KUKA KRL program: EPS_2_26115_ST7256_A_20260223020028.src

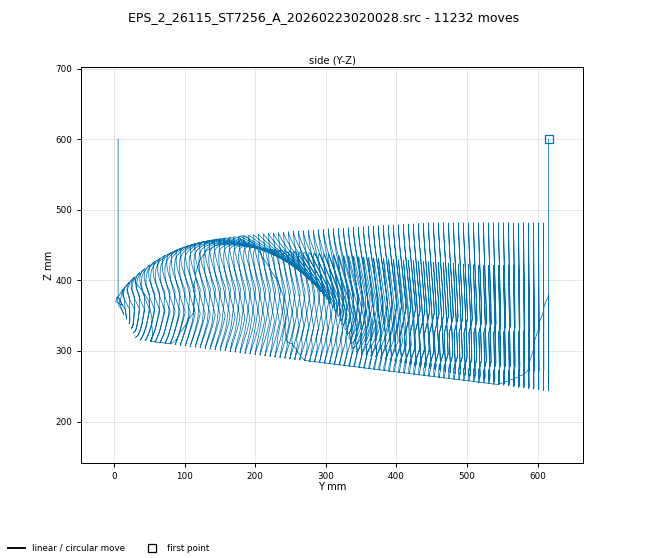
[picture p0: tool path of EPS_2_26115_ST7256_A_20260223020028.src, 11232 of 11234 moves have a stored position in this frame; points joined in program order, loops and branches not executed]
&ACCESS RVP
&REL 4
&COMMENT QRS 19112012
&PARAM EDITMASK = *
DEF PART()
EXT BAS (BAS_COMMAND :IN,REAL :IN )
INT I
BAS (#INITMOV,0 )

;KUKA QRS Post kuka4.cps  Date:22-06-2017 !

File_ID=3070

QRS_PRE_INIT()

;Init var - Until changes are made in qrs_pre_init
Outlet_Square_prg=0
Inlet_1_Square_prg=0
Inlet_2_Square_prg=0
Inlet_3_Square_prg=0
Inlet_4_Square_prg=0
Inlet_5_Square_prg=0

Outlet_1={X 0.000, Y 450.000, Z 332.000, B 0.000, E1 0.000 }
Inlet_1={X 0.000, Y 518.350, Z 272.000, B 0.000, E1 86.000 }
Outlet_1_type=299
Inlet_1_type=299
;QRS#1=Sidecore dimensions
;QRS#2=300-12" PVC SDR 35 Cut Back
;QRS#3=300-12" PVC SDR 35
;QRS#4=
;QRS#5=
;QRS#6=
;QRS#7=
;QRS#8=
;QRS#9=16M PSX
;QRS#10=16M PSX
;QRS#11=
;QRS#12=
;QRS#13=
;QRS#14=
;QRS#15=
;QRS#16=1220x127x762 2,5'
;QRS#17=EPS Height
;QRS#18=481,5
;QRS#19=*
;QRS#20= UPDATED VERSION 22-06-2017
;QRS#21=*
Outlet_Square=0150
Inlet_1_Square=0150
Inlet_2_Square=0
Inlet_3_Square=0
Inlet_4_Square=0
Inlet_5_Square=0
Mill_Square=1
Outlet_Square_Prg=216
Inlet_1_Square_prg=206

QRS_INIT()

$ADVANCE=5

; T1
PTP {E1 173.488,E2 173.488}
PTP {X 0,Y 615.495,A -85,B 0,C 180,E1 173.488,E2 173.488,E3 0,E4 0,E5 0,E6 0}
QRS_SPEED_INIT()
LIN {X 0,Y 615.495,Z 600,A -85,B 0,C 180,E1 173.488,E2 173.488,E3 0,E4 0,E5 0,E6 0} C_VEL
LIN {X 0,Y 615.495,Z 393.639,A -85,B 0,C 180,E1 173.488,E2 173.488} C_VEL
LIN {X 0,Y 615.495,Z 381.654,A -85,B 0,C 180,E1 173.488,E2 173.488} C_VEL
LIN {X 0,Y 615.494,Z 380.114,A -85,B 0,C 180,E1 173.42,E2 173.42} C_VEL
LIN {X 0,Y 615.498,Z 369.133,A -85,B 0,C 180,E1 172.289,E2 172.289} C_VEL
LIN {X 0,Y 615.497,Z 357.594,A -85,B 0,C 180,E1 171.298,E2 171.298} C_VEL
LIN {X 0,Y 615.497,Z 344.878,A -85,B 0,C 180,E1 170.387,E2 170.387} C_VEL
LIN {X 0,Y 615.489,Z 332.281,A -85,B 0,C 180,E1 169.639,E2 169.639} C_VEL
LIN {X 0,Y 615.455,Z 318.443,A -85,B 0,C 180,E1 168.968,E2 168.968} C_VEL
LIN {X 0,Y 615.481,Z 304.474,A -85,B 0,C 180,E1 168.431,E2 168.431} C_VEL
LIN {X 0,Y 615.493,Z 290.197,A -85,B 0,C 180,E1 168.014,E2 168.014} C_VEL
LIN {X 0,Y 615.498,Z 276.029,A -85,B 0,C 180,E1 167.721,E2 167.721} C_VEL
LIN {X 0,Y 615.488,Z 268.934,A -85,B 0,C 180,E1 167.616,E2 167.616} C_VEL
LIN {X 0,Y 615.468,Z 266.187,A -85,B 0,C 180,E1 165.45,E2 165.45} C_VEL
LIN {X 0,Y 615.461,Z 263.623,A -85,B 0,C 180,E1 163.412,E2 163.412} C_VEL
LIN {X 0,Y 615.456,Z 261.066,A -85,B 0,C 180,E1 161.353,E2 161.353} C_VEL
LIN {X 0,Y 615.452,Z 258.516,A -85,B 0,C 180,E1 159.268,E2 159.268} C_VEL
LIN {X 0,Y 615.452,Z 255.973,A -85,B 0,C 180,E1 157.154,E2 157.154} C_VEL
LIN {X 0,Y 615.492,Z 252.76,A -85,B 0,C 180,E1 154.431,E2 154.431} C_VEL
LIN {X 0,Y 615.451,Z 249.501,A -85,B 0,C 180,E1 151.557,E2 151.557} C_VEL
LIN {X 0,Y 615.49,Z 246.653,A -85,B 0,C 180,E1 148.914,E2 148.914} C_VEL
LIN {X 0,Y 615.496,Z 243.464,A -85,B 0,C 180,E1 145.978,E2 145.978} C_VEL
LIN {X 0,Y 615.445,Z 243.325,A -85,B 0,C 180,E1 143.572,E2 143.572} C_VEL
LIN {X 0,Y 615.497,Z 243.315,A -85,B 0,C 180,E1 140.937,E2 140.937} C_VEL
LIN {X 0,Y 615.489,Z 243.322,A -85,B 0,C 180,E1 138.526,E2 138.526} C_VEL
LIN {X 0,Y 615.45,Z 243.325,A -85,B 0,C 180,E1 135.847,E2 135.847} C_VEL
LIN {X 0,Y 615.489,Z 243.315,A -85,B 0,C 180,E1 133.047,E2 133.047} C_VEL
LIN {X 0,Y 615.477,Z 243.327,A -85,B 0,C 180,E1 130.608,E2 130.608} C_VEL
LIN {X 0,Y 615.465,Z 243.325,A -85,B 0,C 180,E1 128.009,E2 128.009} C_VEL
LIN {X 0,Y 615.476,Z 243.319,A -85,B 0,C 180,E1 125.617,E2 125.617} C_VEL
LIN {X 0,Y 615.485,Z 243.325,A -85,B 0,C 180,E1 123.237,E2 123.237} C_VEL
LIN {X 0,Y 615.47,Z 243.32,A -85,B 0,C 180,E1 120.921,E2 120.921} C_VEL
LIN {X 0,Y 615.488,Z 243.325,A -85,B 0,C 180,E1 118.45,E2 118.45} C_VEL
LIN {X 0,Y 615.474,Z 243.325,A -85,B 0,C 180,E1 115.716,E2 115.716} C_VEL
LIN {X 0,Y 615.477,Z 243.321,A -85,B 0,C 180,E1 112.845,E2 112.845} C_VEL
LIN {X 0,Y 615.465,Z 243.324,A -85,B 0,C 180,E1 110.55,E2 110.55} C_VEL
LIN {X 0,Y 615.492,Z 243.325,A -85,B 0,C 180,E1 107.957,E2 107.957} C_VEL
LIN {X 0,Y 615.484,Z 243.32,A -85,B 0,C 180,E1 105.226,E2 105.226} C_VEL
LIN {X 0,Y 615.446,Z 243.325,A -85,B 0,C 180,E1 102.531,E2 102.531} C_VEL
LIN {X 0,Y 615.497,Z 243.316,A -85,B 0,C 180,E1 99.862,E2 99.862} C_VEL
LIN {X 0,Y 615.485,Z 243.328,A -85,B 0,C 180,E1 97.216,E2 97.216} C_VEL
LIN {X 0,Y 615.459,Z 243.325,A -85,B 0,C 180,E1 94.585,E2 94.585} C_VEL
LIN {X 0,Y 615.5,Z 243.313,A -85,B 0,C 180,E1 91.963,E2 91.963} C_VEL
LIN {X 0,Y 615.468,Z 243.325,A -85,B 0,C 180,E1 89.346,E2 89.346} C_VEL
LIN {X 0,Y 615.476,Z 243.326,A -85,B 0,C 180,E1 86.727,E2 86.727} C_VEL
LIN {X 0,Y 615.498,Z 243.314,A -85,B 0,C 180,E1 84.101,E2 84.101} C_VEL
LIN {X 0,Y 615.451,Z 243.325,A -85,B 0,C 180,E1 81.463,E2 81.463} C_VEL
LIN {X 0,Y 615.492,Z 243.322,A -85,B 0,C 180,E1 78.807,E2 78.807} C_VEL
LIN {X 0,Y 615.493,Z 243.322,A -85,B 0,C 180,E1 76.066,E2 76.066} C_VEL
LIN {X 0,Y 615.453,Z 243.324,A -85,B 0,C 180,E1 73.412,E2 73.412} C_VEL
LIN {X 0,Y 615.486,Z 243.316,A -85,B 0,C 180,E1 70.662,E2 70.662} C_VEL
LIN {X 0,Y 615.456,Z 243.325,A -85,B 0,C 180,E1 67.862,E2 67.862} C_VEL
LIN {X 0,Y 615.465,Z 243.322,A -85,B 0,C 180,E1 65.727,E2 65.727} C_VEL
LIN {X 0,Y 615.481,Z 243.324,A -85,B 0,C 180,E1 63.555,E2 63.555} C_VEL
LIN {X 0,Y 615.447,Z 243.325,A -85,B 0,C 180,E1 61.34,E2 61.34} C_VEL
LIN {X 0,Y 615.495,Z 243.319,A -85,B 0,C 180,E1 58.913,E2 58.913} C_VEL
LIN {X 0,Y 615.491,Z 243.318,A -85,B 0,C 180,E1 56.466,E2 56.466} C_VEL
LIN {X 0,Y 615.453,Z 243.325,A -85,B 0,C 180,E1 53.572,E2 53.572} C_VEL
LIN {X 0,Y 615.496,Z 243.314,A -85,B 0,C 180,E1 50.937,E2 50.937} C_VEL
LIN {X 0,Y 615.495,Z 243.326,A -85,B 0,C 180,E1 48.526,E2 48.526} C_VEL
LIN {X 0,Y 615.46,Z 243.325,A -85,B 0,C 180,E1 45.847,E2 45.847} C_VEL
LIN {X 0,Y 615.489,Z 243.316,A -85,B 0,C 180,E1 43.047,E2 43.047} C_VEL
LIN {X 0,Y 615.467,Z 243.325,A -85,B 0,C 180,E1 40.608,E2 40.608} C_VEL
LIN {X 0,Y 615.479,Z 243.325,A -85,B 0,C 180,E1 38.01,E2 38.01} C_VEL
LIN {X 0,Y 615.47,Z 243.32,A -85,B 0,C 180,E1 35.617,E2 35.617} C_VEL
LIN {X 0,Y 615.482,Z 243.328,A -85,B 0,C 180,E1 33.237,E2 33.237} C_VEL
LIN {X 0,Y 615.476,Z 243.318,A -85,B 0,C 180,E1 30.921,E2 30.921} C_VEL
LIN {X 0,Y 615.474,Z 243.324,A -85,B 0,C 180,E1 28.447,E2 28.447} C_VEL
LIN {X 0,Y 615.498,Z 243.323,A -85,B 0,C 180,E1 25.57,E2 25.57} C_VEL
LIN {X 0,Y 615.485,Z 243.322,A -85,B 0,C 180,E1 22.845,E2 22.845} C_VEL
LIN {X 0,Y 615.448,Z 243.326,A -85,B 0,C 180,E1 20.546,E2 20.546} C_VEL
LIN {X 0,Y 615.493,Z 243.324,A -85,B 0,C 180,E1 17.957,E2 17.957} C_VEL
LIN {X 0,Y 615.489,Z 243.321,A -85,B 0,C 180,E1 15.226,E2 15.226} C_VEL
LIN {X 0,Y 615.45,Z 243.325,A -85,B 0,C 180,E1 12.531,E2 12.531} C_VEL
LIN {X 0,Y 615.496,Z 243.314,A -85,B 0,C 180,E1 9.862,E2 9.862} C_VEL
LIN {X 0,Y 615.476,Z 243.326,A -85,B 0,C 180,E1 7.216,E2 7.216} C_VEL
LIN {X 0,Y 615.471,Z 243.325,A -85,B 0,C 180,E1 4.585,E2 4.585} C_VEL
LIN {X 0,Y 615.5,Z 243.313,A -85,B 0,C 180,E1 1.963,E2 1.963} C_VEL
LIN {X 0,Y 615.456,Z 243.325,A -85,B 0,C 180,E1 -0.654,E2 -0.654} C_VEL
LIN {X 0,Y 615.488,Z 243.328,A -85,B 0,C 180,E1 -3.273,E2 -3.273} C_VEL
LIN {X 0,Y 615.499,Z 243.316,A -85,B 0,C 180,E1 -5.898,E2 -5.898} C_VEL
LIN {X 0,Y 615.446,Z 243.325,A -85,B 0,C 180,E1 -8.537,E2 -8.537} C_VEL
LIN {X 0,Y 615.484,Z 243.321,A -85,B 0,C 180,E1 -11.193,E2 -11.193} C_VEL
LIN {X 0,Y 615.498,Z 243.325,A -85,B 0,C 180,E1 -13.935,E2 -13.935} C_VEL
LIN {X 0,Y 615.466,Z 243.324,A -85,B 0,C 180,E1 -16.587,E2 -16.587} C_VEL
LIN {X 0,Y 615.482,Z 243.317,A -85,B 0,C 180,E1 -19.338,E2 -19.338} C_VEL
LIN {X 0,Y 615.448,Z 243.325,A -85,B 0,C 180,E1 -22.138,E2 -22.138} C_VEL
LIN {X 0,Y 615.477,Z 243.322,A -85,B 0,C 180,E1 -24.272,E2 -24.272} C_VEL
LIN {X 0,Y 615.468,Z 243.321,A -85,B 0,C 180,E1 -27.041,E2 -27.041} C_VEL
LIN {X 0,Y 615.464,Z 243.321,A -85,B 0,C 180,E1 -29.79,E2 -29.79} C_VEL
LIN {X 0,Y 615.481,Z 243.323,A -85,B 0,C 180,E1 -32.458,E2 -32.458} C_VEL
LIN {X 0,Y 615.459,Z 243.325,A -85,B 0,C 180,E1 -34.817,E2 -34.817} C_VEL
LIN {X 0,Y 615.492,Z 243.316,A -85,B 0,C 180,E1 -37.242,E2 -37.242} C_VEL
LIN {X 0,Y 615.474,Z 243.324,A -85,B 0,C 180,E1 -40.087,E2 -40.087} C_VEL
LIN {X 0,Y 615.451,Z 243.325,A -85,B 0,C 180,E1 -42.356,E2 -42.356} C_VEL
LIN {X 0,Y 615.491,Z 243.315,A -85,B 0,C 180,E1 -45.068,E2 -45.068} C_VEL
LIN {X 0,Y 615.454,Z 243.325,A -85,B 0,C 180,E1 -47.923,E2 -47.923} C_VEL
LIN {X 0,Y 615.474,Z 243.517,A -85,B 0,C 180,E1 -48.715,E2 -48.715} C_VEL
LIN {X 0,Y 615.44,Z 251.638,A -85,B 0,C 180,E1 -51.511,E2 -51.511} C_VEL
LIN {X 0,Y 615.45,Z 257.822,A -85,B 0,C 180,E1 -53.572,E2 -53.572} C_VEL
LIN {X 0,Y 615.483,Z 265.237,A -85,B 0,C 180,E1 -55.977,E2 -55.977} C_VEL
LIN {X 0,Y 615.485,Z 274.588,A -85,B 0,C 180,E1 -58.914,E2 -58.914} C_VEL
LIN {X 0,Y 615.486,Z 283.218,A -85,B 0,C 180,E1 -61.55,E2 -61.55} C_VEL
LIN {X 0,Y 615.472,Z 292.408,A -85,B 0,C 180,E1 -64.283,E2 -64.283} C_VEL
LIN {X 0,Y 615.455,Z 302.27,A -85,B 0,C 180,E1 -67.154,E2 -67.154} C_VEL
LIN {X 0,Y 615.425,Z 310.351,A -85,B 0,C 180,E1 -69.459,E2 -69.459} C_VEL
LIN {X 0,Y 615.486,Z 319.519,A -85,B 0,C 180,E1 -72.043,E2 -72.043} C_VEL
LIN {X 0,Y 615.465,Z 325.159,A -85,B 0,C 180,E1 -73.609,E2 -73.609} C_VEL
LIN {X 0,Y 615.49,Z 343.311,A -85,B 0,C 180,E1 -73.901,E2 -73.901} C_VEL
LIN {X 0,Y 615.497,Z 357.798,A -85,B 0,C 180,E1 -74.265,E2 -74.265} C_VEL
LIN {X 0,Y 615.463,Z 372.664,A -85,B 0,C 180,E1 -74.773,E2 -74.773} C_VEL
LIN {X 0,Y 615.468,Z 386.103,A -85,B 0,C 180,E1 -75.366,E2 -75.366} C_VEL
LIN {X 0,Y 615.498,Z 400.008,A -85,B 0,C 180,E1 -76.126,E2 -76.126} C_VEL
LIN {X 0,Y 615.496,Z 412.63,A -85,B 0,C 180,E1 -76.967,E2 -76.967} C_VEL
LIN {X 0,Y 615.496,Z 423.227,A -85,B 0,C 180,E1 -77.805,E2 -77.805} C_VEL
LIN {X 0,Y 615.496,Z 433.973,A -85,B 0,C 180,E1 -78.807,E2 -78.807} C_VEL
LIN {X 0,Y 615.496,Z 444.421,A -85,B 0,C 180,E1 -79.972,E2 -79.972} C_VEL
LIN {X 0,Y 615.496,Z 453.101,A -85,B 0,C 180,E1 -81.132,E2 -81.132} C_VEL
LIN {X 0,Y 615.494,Z 461.224,A -85,B 0,C 180,E1 -82.454,E2 -82.454} C_VEL
LIN {X 0,Y 615.496,Z 467.729,A -85,B 0,C 180,E1 -83.773,E2 -83.773} C_VEL
LIN {X 0,Y 615.496,Z 472.809,A -85,B 0,C 180,E1 -85.087,E2 -85.087} C_VEL
LIN {X 0,Y 615.495,Z 475.74,A -85,B 0,C 180,E1 -86.071,E2 -86.071} C_VEL
LIN {X 0,Y 615.494,Z 478.6,A -85,B 0,C 180,E1 -87.382,E2 -87.382} C_VEL
LIN {X 0,Y 615.492,Z 480.307,A -85,B 0,C 180,E1 -88.691,E2 -88.691} C_VEL
LIN {X 0,Y 615.491,Z 480.889,A -85,B 0,C 180,E1 -90,E2 -90} C_VEL
LIN {X 0,Y 615.492,Z 480.307,A -85,B 0,C 180,E1 -91.309,E2 -91.309} C_VEL
LIN {X 0,Y 615.494,Z 478.6,A -85,B 0,C 180,E1 -92.618,E2 -92.618} C_VEL
LIN {X 0,Y 615.495,Z 475.74,A -85,B 0,C 180,E1 -93.928,E2 -93.928} C_VEL
LIN {X 0,Y 615.491,Z 471.666,A -85,B 0,C 180,E1 -95.241,E2 -95.241} C_VEL
LIN {X 0,Y 615.49,Z 466.159,A -85,B 0,C 180,E1 -96.58,E2 -96.58} C_VEL
LIN {X 0,Y 615.493,Z 459.393,A -85,B 0,C 180,E1 -97.876,E2 -97.876} C_VEL
LIN {X 0,Y 615.495,Z 450.808,A -85,B 0,C 180,E1 -99.199,E2 -99.199} C_VEL
LIN {X 0,Y 615.494,Z 441.666,A -85,B 0,C 180,E1 -100.361,E2 -100.361} C_VEL
LIN {X 0,Y 615.497,Z 432.353,A -85,B 0,C 180,E1 -101.36,E2 -101.36} C_VEL
LIN {X 0,Y 615.496,Z 421.292,A -85,B 0,C 180,E1 -102.363,E2 -102.363} C_VEL
LIN {X 0,Y 615.498,Z 409.151,A -85,B 0,C 180,E1 -103.285,E2 -103.285} C_VEL
LIN {X 0,Y 615.498,Z 396.404,A -85,B 0,C 180,E1 -104.09,E2 -104.09} C_VEL
LIN {X 0,Y 615.46,Z 382.609,A -85,B 0,C 180,E1 -104.803,E2 -104.803} C_VEL
LIN {X 0,Y 615.474,Z 368.18,A -85,B 0,C 180,E1 -105.396,E2 -105.396} C_VEL
LIN {X 0,Y 615.496,Z 353.245,A -85,B 0,C 180,E1 -105.863,E2 -105.863} C_VEL
LIN {X 0,Y 615.483,Z 338.115,A -85,B 0,C 180,E1 -106.196,E2 -106.196} C_VEL
LIN {X 0,Y 615.465,Z 325.159,A -85,B 0,C 180,E1 -106.391,E2 -106.391} C_VEL
LIN {X 0,Y 615.433,Z 317.07,A -85,B 0,C 180,E1 -108.648,E2 -108.648} C_VEL
LIN {X 0,Y 615.498,Z 307.197,A -85,B 0,C 180,E1 -111.432,E2 -111.432} C_VEL
LIN {X 0,Y 615.446,Z 297.341,A -85,B 0,C 180,E1 -114.274,E2 -114.274} C_VEL
LIN {X 0,Y 615.491,Z 287.908,A -85,B 0,C 180,E1 -117.046,E2 -117.046} C_VEL
LIN {X 0,Y 615.477,Z 278.794,A -85,B 0,C 180,E1 -119.793,E2 -119.793} C_VEL
LIN {X 0,Y 615.476,Z 270.181,A -85,B 0,C 180,E1 -122.458,E2 -122.458} C_VEL
LIN {X 0,Y 615.493,Z 261.529,A -85,B 0,C 180,E1 -125.214,E2 -125.214} C_VEL
LIN {X 0,Y 615.446,Z 253.069,A -85,B 0,C 180,E1 -128.007,E2 -128.007} C_VEL
LIN {X 0,Y 615.427,Z 246.977,A -85,B 0,C 180,E1 -130.082,E2 -130.082} C_VEL
LIN {X 0,Y 615.46,Z 243.324,A -85,B 0,C 180,E1 -131.381,E2 -131.381} C_VEL
LIN {X 0,Y 615.44,Z 243.322,A -85,B 0,C 180,E1 -133.993,E2 -133.993} C_VEL
LIN {X 0,Y 615.456,Z 243.322,A -85,B 0,C 180,E1 -136.006,E2 -136.006} C_VEL
LIN {X 0,Y 615.467,Z 243.321,A -85,B 0,C 180,E1 -137.922,E2 -137.922} C_VEL
LIN {X 0,Y 615.493,Z 246.192,A -85,B 0,C 180,E1 -140.25,E2 -140.25} C_VEL
LIN {X 0,Y 615.487,Z 249.063,A -85,B 0,C 180,E1 -143.064,E2 -143.064} C_VEL
LIN {X 0,Y 615.458,Z 251.362,A -85,B 0,C 180,E1 -145.304,E2 -145.304} C_VEL
LIN {X 0,Y 615.461,Z 254.12,A -85,B 0,C 180,E1 -147.674,E2 -147.674} C_VEL
LIN {X 0,Y 615.489,Z 257.579,A -85,B 0,C 180,E1 -150.594,E2 -150.594} C_VEL
LIN {X 0,Y 615.465,Z 260.463,A -85,B 0,C 180,E1 -152.96,E2 -152.96} C_VEL
LIN {X 0,Y 615.481,Z 263.903,A -85,B 0,C 180,E1 -155.728,E2 -155.728} C_VEL
LIN {X 0,Y 615.49,Z 267.47,A -85,B 0,C 180,E1 -158.568,E2 -158.568} C_VEL
LIN {X 0,Y 615.483,Z 268.939,A -85,B 0,C 180,E1 -159.709,E2 -159.709} C_VEL
LIN {X 0,Y 615.491,Z 284.345,A -85,B 0,C 180,E1 -159.967,E2 -159.967} C_VEL
LIN {X 0,Y 615.489,Z 299.504,A -85,B 0,C 180,E1 -160.359,E2 -160.359} C_VEL
LIN {X 0,Y 615.464,Z 314.236,A -85,B 0,C 180,E1 -160.878,E2 -160.878} C_VEL
LIN {X 0,Y 615.481,Z 329.195,A -85,B 0,C 180,E1 -161.563,E2 -161.563} C_VEL
LIN {X 0,Y 615.498,Z 342.188,A -85,B 0,C 180,E1 -162.301,E2 -162.301} C_VEL
LIN {X 0,Y 615.496,Z 354.643,A -85,B 0,C 180,E1 -163.158,E2 -163.158} C_VEL
LIN {X 0,Y 615.496,Z 366.064,A -85,B 0,C 180,E1 -164.095,E2 -164.095} C_VEL
LIN {X 0,Y 615.494,Z 376.512,A -85,B 0,C 180,E1 -165.113,E2 -165.113} C_VEL
LIN {X 0,Y 615.493,Z 386.686,A -85,B 0,C 180,E1 -166.294,E2 -166.294} C_VEL
LIN {X 0,Y 615.493,Z 395.074,A -85,B 0,C 180,E1 -167.47,E2 -167.47} C_VEL
LIN {X 0,Y 615.495,Z 402.907,A -85,B 0,C 180,E1 -168.807,E2 -168.807} C_VEL
LIN {X 0,Y 615.498,Z 409.106,A -85,B 0,C 180,E1 -170.138,E2 -170.138} C_VEL
LIN {X 0,Y 615.491,Z 413.87,A -85,B 0,C 180,E1 -171.464,E2 -171.464} C_VEL
LIN {X 0,Y 615.493,Z 417.345,A -85,B 0,C 180,E1 -172.785,E2 -172.785} C_VEL
LIN {X 0,Y 615.499,Z 419.616,A -85,B 0,C 180,E1 -174.102,E2 -174.102} C_VEL
LIN {X 0,Y 615.497,Z 420.745,A -85,B 0,C 180,E1 -175.416,E2 -175.416} C_VEL
LIN {X 0,Y 615.491,Z 420.734,A -85,B 0,C 180,E1 -176.727,E2 -176.727} C_VEL
LIN {X 0,Y 615.5,Z 419.559,A -85,B 0,C 180,E1 -178.037,E2 -178.037} C_VEL
LIN {X 0,Y 615.491,Z 417.258,A -85,B 0,C 180,E1 -179.346,E2 -179.346} C_VEL
LIN {X 0,Y 615.49,Z 413.781,A -85,B 0,C 180,E1 -180.654,E2 -180.654} C_VEL
LIN {X 0,Y 615.5,Z 409.056,A -85,B 0,C 180,E1 -181.963,E2 -181.963} C_VEL
LIN {X 0,Y 615.492,Z 402.961,A -85,B 0,C 180,E1 -183.273,E2 -183.273} C_VEL
LIN {X 0,Y 615.494,Z 395.311,A -85,B 0,C 180,E1 -184.585,E2 -184.585} C_VEL
LIN {X 0,Y 615.495,Z 387.166,A -85,B 0,C 180,E1 -185.734,E2 -185.734} C_VEL
LIN {X 0,Y 615.494,Z 380.114,A -85,B 0,C 180,E1 -186.58,E2 -186.58} C_VEL
LIN {X 0,Y 614.823,Z 376.463,A -85,B 0,C 180,E1 -187.003,E2 -187.003} C_VEL
LIN {X 0,Y 611.954,Z 370.281,A -85,B 0,C 180,E1 -187.683,E2 -187.683} C_VEL
LIN {X 0,Y 609.129,Z 363.784,A -85,B 0,C 180,E1 -188.335,E2 -188.335} C_VEL
LIN {X 0,Y 608.527,Z 359.446,A -85,B 0,C 180,E1 -188.708,E2 -188.708} C_VEL
LIN {X 0,Y 608.536,Z 346.882,A -85,B 0,C 180,E1 -189.64,E2 -189.64} C_VEL
LIN {X 0,Y 608.57,Z 333.16,A -85,B 0,C 180,E1 -190.48,E2 -190.48} C_VEL
LIN {X 0,Y 608.559,Z 318.892,A -85,B 0,C 180,E1 -191.187,E2 -191.187} C_VEL
LIN {X 0,Y 608.62,Z 304.623,A -85,B 0,C 180,E1 -191.743,E2 -191.743} C_VEL
LIN {X 0,Y 608.667,Z 289.52,A -85,B 0,C 180,E1 -192.186,E2 -192.186} C_VEL
LIN {X 0,Y 608.694,Z 274.921,A -85,B 0,C 180,E1 -192.482,E2 -192.482} C_VEL
LIN {X 0,Y 608.431,Z 269.386,A -85,B 0,C 180,E1 -192.572,E2 -192.572} C_VEL
LIN {X 0,Y 608.399,Z 266.664,A -85,B 0,C 180,E1 -194.723,E2 -194.723} C_VEL
LIN {X 0,Y 608.399,Z 264.085,A -85,B 0,C 180,E1 -196.786,E2 -196.786} C_VEL
LIN {X 0,Y 608.409,Z 260.656,A -85,B 0,C 180,E1 -199.572,E2 -199.572} C_VEL
LIN {X 0,Y 608.398,Z 257.178,A -85,B 0,C 180,E1 -202.461,E2 -202.461} C_VEL
LIN {X 0,Y 608.404,Z 254.689,A -85,B 0,C 180,E1 -204.573,E2 -204.573} C_VEL
LIN {X 0,Y 608.416,Z 251.668,A -85,B 0,C 180,E1 -207.195,E2 -207.195} C_VEL
LIN {X 0,Y 608.422,Z 248.679,A -85,B 0,C 180,E1 -209.963,E2 -209.963} C_VEL
LIN {X 0,Y 608.436,Z 245.927,A -85,B 0,C 180,E1 -212.518,E2 -212.518} C_VEL
LIN {X 0,Y 608.452,Z 244.611,A -85,B 0,C 180,E1 -213.731,E2 -213.731} C_VEL
LIN {X 0,Y 608.44,Z 244.321,A -85,B 0,C 180,E1 -215.278,E2 -215.278} C_VEL
LIN {X 0,Y 608.449,Z 244.317,A -85,B 0,C 180,E1 -217.748,E2 -217.748} C_VEL
LIN {X 0,Y 608.453,Z 244.32,A -85,B 0,C 180,E1 -220.329,E2 -220.329} C_VEL
LIN {X 0,Y 608.477,Z 244.318,A -85,B 0,C 180,E1 -223.309,E2 -223.309} C_VEL
LIN {X 0,Y 608.464,Z 244.32,A -85,B 0,C 180,E1 -226.13,E2 -226.13} C_VEL
LIN {X 0,Y 608.454,Z 244.318,A -85,B 0,C 180,E1 -228.823,E2 -228.823} C_VEL
LIN {X 0,Y 608.449,Z 244.318,A -85,B 0,C 180,E1 -231.762,E2 -231.762} C_VEL
LIN {X 0,Y 608.447,Z 244.322,A -85,B 0,C 180,E1 -233.955,E2 -233.955} C_VEL
LIN {X 0,Y 608.446,Z 244.318,A -85,B 0,C 180,E1 -236.328,E2 -236.328} C_VEL
LIN {X 0,Y 608.448,Z 244.32,A -85,B 0,C 180,E1 -238.733,E2 -238.733} C_VEL
LIN {X 0,Y 608.473,Z 244.32,A -85,B 0,C 180,E1 -241.381,E2 -241.381} C_VEL
LIN {X 0,Y 608.425,Z 244.321,A -85,B 0,C 180,E1 -243.963,E2 -243.963} C_VEL
LIN {X 0,Y 608.449,Z 244.317,A -85,B 0,C 180,E1 -246.876,E2 -246.876} C_VEL
LIN {X 0,Y 608.454,Z 244.319,A -85,B 0,C 180,E1 -249.326,E2 -249.326} C_VEL
LIN {X 0,Y 608.439,Z 244.321,A -85,B 0,C 180,E1 -251.828,E2 -251.828} C_VEL
LIN {X 0,Y 608.47,Z 244.315,A -85,B 0,C 180,E1 -254.594,E2 -254.594} C_VEL
LIN {X 0,Y 608.422,Z 244.321,A -85,B 0,C 180,E1 -257.322,E2 -257.322} C_VEL
LIN {X 0,Y 608.462,Z 244.318,A -85,B 0,C 180,E1 -260.023,E2 -260.023} C_VEL
LIN {X 0,Y 608.465,Z 244.321,A -85,B 0,C 180,E1 -262.701,E2 -262.701} C_VEL
LIN {X 0,Y 608.426,Z 244.321,A -85,B 0,C 180,E1 -265.362,E2 -265.362} C_VEL
LIN {X 0,Y 608.47,Z 244.315,A -85,B 0,C 180,E1 -268.014,E2 -268.014} C_VEL
LIN {X 0,Y 608.465,Z 244.318,A -85,B 0,C 180,E1 -270.662,E2 -270.662} C_VEL
LIN {X 0,Y 608.471,Z 244.319,A -85,B 0,C 180,E1 -273.311,E2 -273.311} C_VEL
LIN {X 0,Y 608.471,Z 244.315,A -85,B 0,C 180,E1 -275.967,E2 -275.967} C_VEL
LIN {X 0,Y 608.427,Z 244.32,A -85,B 0,C 180,E1 -278.637,E2 -278.637} C_VEL
LIN {X 0,Y 608.482,Z 244.316,A -85,B 0,C 180,E1 -281.324,E2 -281.324} C_VEL
LIN {X 0,Y 608.473,Z 244.32,A -85,B 0,C 180,E1 -284.037,E2 -284.037} C_VEL
LIN {X 0,Y 608.432,Z 244.321,A -85,B 0,C 180,E1 -286.785,E2 -286.785} C_VEL
LIN {X 0,Y 608.454,Z 244.317,A -85,B 0,C 180,E1 -289.571,E2 -289.571} C_VEL
LIN {X 0,Y 608.433,Z 244.319,A -85,B 0,C 180,E1 -292.469,E2 -292.469} C_VEL
LIN {X 0,Y 608.453,Z 244.317,A -85,B 0,C 180,E1 -295.301,E2 -295.301} C_VEL
LIN {X 0,Y 608.446,Z 244.32,A -85,B 0,C 180,E1 -297.518,E2 -297.518} C_VEL
LIN {X 0,Y 608.441,Z 244.321,A -85,B 0,C 180,E1 -300.547,E2 -300.547} C_VEL
LIN {X 0,Y 608.463,Z 244.316,A -85,B 0,C 180,E1 -302.88,E2 -302.88} C_VEL
LIN {X 0,Y 608.43,Z 244.324,A -85,B 0,C 180,E1 -305.279,E2 -305.279} C_VEL
LIN {X 0,Y 608.459,Z 244.316,A -85,B 0,C 180,E1 -307.747,E2 -307.747} C_VEL
LIN {X 0,Y 608.446,Z 244.32,A -85,B 0,C 180,E1 -310.328,E2 -310.328} C_VEL
LIN {X 0,Y 608.445,Z 244.323,A -85,B 0,C 180,E1 -312.961,E2 -312.961} C_VEL
LIN {X 0,Y 608.454,Z 244.319,A -85,B 0,C 180,E1 -315.737,E2 -315.737} C_VEL
LIN {X 0,Y 608.453,Z 244.318,A -85,B 0,C 180,E1 -318.659,E2 -318.659} C_VEL
LIN {X 0,Y 608.46,Z 244.317,A -85,B 0,C 180,E1 -321.761,E2 -321.761} C_VEL
LIN {X 0,Y 608.446,Z 244.32,A -85,B 0,C 180,E1 -323.955,E2 -323.955} C_VEL
LIN {X 0,Y 608.448,Z 244.319,A -85,B 0,C 180,E1 -326.328,E2 -326.328} C_VEL
LIN {X 0,Y 608.451,Z 244.318,A -85,B 0,C 180,E1 -328.733,E2 -328.733} C_VEL
LIN {X 0,Y 608.47,Z 244.32,A -85,B 0,C 180,E1 -331.382,E2 -331.382} C_VEL
LIN {X 0,Y 608.432,Z 244.321,A -85,B 0,C 180,E1 -333.964,E2 -333.964} C_VEL
LIN {X 0,Y 608.473,Z 244.317,A -85,B 0,C 180,E1 -336.155,E2 -336.155} C_VEL
LIN {X 0,Y 608.447,Z 244.322,A -85,B 0,C 180,E1 -339.018,E2 -339.018} C_VEL
LIN {X 0,Y 608.442,Z 244.323,A -85,B 0,C 180,E1 -341.828,E2 -341.828} C_VEL
LIN {X 0,Y 608.473,Z 244.316,A -85,B 0,C 180,E1 -344.594,E2 -344.594} C_VEL
LIN {X 0,Y 608.421,Z 244.321,A -85,B 0,C 180,E1 -347.322,E2 -347.322} C_VEL
LIN {X 0,Y 608.465,Z 244.316,A -85,B 0,C 180,E1 -350.023,E2 -350.023} C_VEL
LIN {X 0,Y 608.444,Z 244.323,A -85,B 0,C 180,E1 -352.7,E2 -352.7} C_VEL
LIN {X 0,Y 608.437,Z 244.321,A -85,B 0,C 180,E1 -355.362,E2 -355.362} C_VEL
LIN {X 0,Y 608.469,Z 244.315,A -85,B 0,C 180,E1 -358.014,E2 -358.014} C_VEL
LIN {X 0,Y 608.454,Z 244.318,A -85,B 0,C 180,E1 -360.662,E2 -360.662} C_VEL
LIN {X 0,Y 608.482,Z 244.319,A -85,B 0,C 180,E1 -363.311,E2 -363.311} C_VEL
LIN {X 0,Y 608.469,Z 244.317,A -85,B 0,C 180,E1 -365.967,E2 -365.967} C_VEL
LIN {X 0,Y 608.426,Z 244.32,A -85,B 0,C 180,E1 -368.636,E2 -368.636} C_VEL
LIN {X 0,Y 608.462,Z 244.317,A -85,B 0,C 180,E1 -371.324,E2 -371.324} C_VEL
LIN {X 0,Y 608.475,Z 244.319,A -85,B 0,C 180,E1 -374.037,E2 -374.037} C_VEL
LIN {X 0,Y 608.438,Z 244.322,A -85,B 0,C 180,E1 -376.784,E2 -376.784} C_VEL
LIN {X 0,Y 608.451,Z 244.318,A -85,B 0,C 180,E1 -379.57,E2 -379.57} C_VEL
LIN {X 0,Y 608.433,Z 244.32,A -85,B 0,C 180,E1 -382.469,E2 -382.469} C_VEL
LIN {X 0,Y 608.449,Z 244.324,A -85,B 0,C 180,E1 -384.571,E2 -384.571} C_VEL
LIN {X 0,Y 608.471,Z 244.316,A -85,B 0,C 180,E1 -387.205,E2 -387.205} C_VEL
LIN {X 0,Y 608.43,Z 244.32,A -85,B 0,C 180,E1 -389.964,E2 -389.964} C_VEL
LIN {X 0,Y 608.458,Z 244.318,A -85,B 0,C 180,E1 -392.521,E2 -392.521} C_VEL
LIN {X 0,Y 608.424,Z 244.322,A -85,B 0,C 180,E1 -394.901,E2 -394.901} C_VEL
LIN {X 0,Y 608.467,Z 244.316,A -85,B 0,C 180,E1 -397.746,E2 -397.746} C_VEL
LIN {X 0,Y 608.435,Z 244.32,A -85,B 0,C 180,E1 -400.327,E2 -400.327} C_VEL
LIN {X 0,Y 608.467,Z 244.316,A -85,B 0,C 180,E1 -403.308,E2 -403.308} C_VEL
LIN {X 0,Y 608.473,Z 244.318,A -85,B 0,C 180,E1 -406.13,E2 -406.13} C_VEL
LIN {X 0,Y 608.44,Z 244.337,A -85,B 0,C 180,E1 -408.425,E2 -408.425} C_VEL
LIN {X 0,Y 608.541,Z 250.775,A -85,B 0,C 180,E1 -410.694,E2 -410.694} C_VEL
LIN {X 0,Y 608.507,Z 259.067,A -85,B 0,C 180,E1 -413.501,E2 -413.501} C_VEL
LIN {X 0,Y 608.519,Z 266.495,A -85,B 0,C 180,E1 -415.934,E2 -415.934} C_VEL
LIN {X 0,Y 608.491,Z 275.29,A -85,B 0,C 180,E1 -418.726,E2 -418.726} C_VEL
LIN {X 0,Y 608.499,Z 283.878,A -85,B 0,C 180,E1 -421.376,E2 -421.376} C_VEL
LIN {X 0,Y 608.447,Z 292.488,A -85,B 0,C 180,E1 -423.964,E2 -423.964} C_VEL
LIN {X 0,Y 608.472,Z 301.153,A -85,B 0,C 180,E1 -426.516,E2 -426.516} C_VEL
LIN {X 0,Y 608.42,Z 310.923,A -85,B 0,C 180,E1 -429.333,E2 -429.333} C_VEL
LIN {X 0,Y 608.45,Z 320.958,A -85,B 0,C 180,E1 -432.176,E2 -432.176} C_VEL
LIN {X 0,Y 608.426,Z 325.415,A -85,B 0,C 180,E1 -433.422,E2 -433.422} C_VEL
LIN {X 0,Y 608.682,Z 332.489,A -85,B 0,C 180,E1 -433.528,E2 -433.528} C_VEL
LIN {X 0,Y 608.675,Z 347.584,A -85,B 0,C 180,E1 -433.814,E2 -433.814} C_VEL
LIN {X 0,Y 608.623,Z 363.2,A -85,B 0,C 180,E1 -434.254,E2 -434.254} C_VEL
LIN {X 0,Y 608.573,Z 376.817,A -85,B 0,C 180,E1 -434.768,E2 -434.768} C_VEL
LIN {X 0,Y 608.565,Z 391.1,A -85,B 0,C 180,E1 -435.453,E2 -435.453} C_VEL
LIN {X 0,Y 608.558,Z 404.109,A -85,B 0,C 180,E1 -436.22,E2 -436.22} C_VEL
LIN {X 0,Y 608.518,Z 416.103,A -85,B 0,C 180,E1 -437.069,E2 -437.069} C_VEL
LIN {X 0,Y 608.509,Z 427.191,A -85,B 0,C 180,E1 -438.001,E2 -438.001} C_VEL
LIN {X 0,Y 608.477,Z 437.641,A -85,B 0,C 180,E1 -439.04,E2 -439.04} C_VEL
LIN {X 0,Y 608.471,Z 447.368,A -85,B 0,C 180,E1 -440.191,E2 -440.191} C_VEL
LIN {X 0,Y 608.467,Z 455.654,A -85,B 0,C 180,E1 -441.364,E2 -441.364} C_VEL
LIN {X 0,Y 608.456,Z 463.426,A -85,B 0,C 180,E1 -442.7,E2 -442.7} C_VEL
LIN {X 0,Y 608.437,Z 469.608,A -85,B 0,C 180,E1 -444.033,E2 -444.033} C_VEL
LIN {X 0,Y 608.427,Z 474.383,A -85,B 0,C 180,E1 -445.362,E2 -445.362} C_VEL
LIN {X 0,Y 608.421,Z 477.885,A -85,B 0,C 180,E1 -446.689,E2 -446.689} C_VEL
LIN {X 0,Y 608.444,Z 480.191,A -85,B 0,C 180,E1 -448.014,E2 -448.014} C_VEL
LIN {X 0,Y 608.434,Z 481.351,A -85,B 0,C 180,E1 -449.338,E2 -449.338} C_VEL
LIN {X 0,Y 608.434,Z 481.351,A -85,B 0,C 180,E1 -450.662,E2 -450.662} C_VEL
LIN {X 0,Y 608.444,Z 480.191,A -85,B 0,C 180,E1 -451.986,E2 -451.986} C_VEL
LIN {X 0,Y 608.421,Z 477.885,A -85,B 0,C 180,E1 -453.311,E2 -453.311} C_VEL
LIN {X 0,Y 608.427,Z 474.383,A -85,B 0,C 180,E1 -454.638,E2 -454.638} C_VEL
LIN {X 0,Y 608.437,Z 469.608,A -85,B 0,C 180,E1 -455.967,E2 -455.967} C_VEL
LIN {X 0,Y 608.456,Z 463.426,A -85,B 0,C 180,E1 -457.3,E2 -457.3} C_VEL
LIN {X 0,Y 608.467,Z 455.654,A -85,B 0,C 180,E1 -458.636,E2 -458.636} C_VEL
LIN {X 0,Y 608.471,Z 447.369,A -85,B 0,C 180,E1 -459.809,E2 -459.809} C_VEL
LIN {X 0,Y 608.492,Z 436.653,A -85,B 0,C 180,E1 -461.063,E2 -461.063} C_VEL
LIN {X 0,Y 608.522,Z 425.275,A -85,B 0,C 180,E1 -462.168,E2 -462.168} C_VEL
LIN {X 0,Y 608.547,Z 413.853,A -85,B 0,C 180,E1 -463.1,E2 -463.1} C_VEL
LIN {X 0,Y 608.563,Z 401.446,A -85,B 0,C 180,E1 -463.95,E2 -463.95} C_VEL
LIN {X 0,Y 608.576,Z 387.858,A -85,B 0,C 180,E1 -464.718,E2 -464.718} C_VEL
LIN {X 0,Y 608.593,Z 373.791,A -85,B 0,C 180,E1 -465.36,E2 -465.36} C_VEL
LIN {X 0,Y 608.643,Z 359.295,A -85,B 0,C 180,E1 -465.874,E2 -465.874} C_VEL
LIN {X 0,Y 608.675,Z 343.318,A -85,B 0,C 180,E1 -466.284,E2 -466.284} C_VEL
LIN {X 0,Y 608.671,Z 327.102,A -85,B 0,C 180,E1 -466.546,E2 -466.546} C_VEL
LIN {X 0,Y 608.433,Z 325.333,A -85,B 0,C 180,E1 -466.6,E2 -466.6} C_VEL
LIN {X 0,Y 608.435,Z 316.007,A -85,B 0,C 180,E1 -469.22,E2 -469.22} C_VEL
LIN {X 0,Y 608.445,Z 306.105,A -85,B 0,C 180,E1 -472.049,E2 -472.049} C_VEL
LIN {X 0,Y 608.439,Z 297.44,A -85,B 0,C 180,E1 -474.572,E2 -474.572} C_VEL
LIN {X 0,Y 608.484,Z 288.561,A -85,B 0,C 180,E1 -477.208,E2 -477.208} C_VEL
LIN {X 0,Y 608.484,Z 279.477,A -85,B 0,C 180,E1 -479.974,E2 -479.974} C_VEL
LIN {X 0,Y 608.516,Z 271.296,A -85,B 0,C 180,E1 -482.531,E2 -482.531} C_VEL
LIN {X 0,Y 608.553,Z 262.781,A -85,B 0,C 180,E1 -485.271,E2 -485.271} C_VEL
LIN {X 0,Y 608.532,Z 255.354,A -85,B 0,C 180,E1 -487.742,E2 -487.742} C_VEL
LIN {X 0,Y 608.517,Z 247.82,A -85,B 0,C 180,E1 -490.336,E2 -490.336} C_VEL
LIN {X 0,Y 608.426,Z 244.322,A -85,B 0,C 180,E1 -491.624,E2 -491.624} C_VEL
LIN {X 0,Y 608.425,Z 244.321,A -85,B 0,C 180,E1 -494.261,E2 -494.261} C_VEL
LIN {X 0,Y 608.45,Z 244.317,A -85,B 0,C 180,E1 -497.04,E2 -497.04} C_VEL
LIN {X 0,Y 608.448,Z 244.32,A -85,B 0,C 180,E1 -497.938,E2 -497.938} C_VEL
LIN {X 0,Y 608.45,Z 247.646,A -85,B 0,C 180,E1 -500.705,E2 -500.705} C_VEL
LIN {X 0,Y 608.447,Z 250.017,A -85,B 0,C 180,E1 -503.085,E2 -503.085} C_VEL
LIN {X 0,Y 608.396,Z 252.389,A -85,B 0,C 180,E1 -505.526,E2 -505.526} C_VEL
LIN {X 0,Y 608.404,Z 255.14,A -85,B 0,C 180,E1 -507.902,E2 -507.902} C_VEL
LIN {X 0,Y 608.444,Z 257.88,A -85,B 0,C 180,E1 -510.219,E2 -510.219} C_VEL
LIN {X 0,Y 608.418,Z 261.005,A -85,B 0,C 180,E1 -512.805,E2 -512.805} C_VEL
LIN {X 0,Y 608.412,Z 264.237,A -85,B 0,C 180,E1 -515.427,E2 -515.427} C_VEL
LIN {X 0,Y 608.416,Z 267.849,A -85,B 0,C 180,E1 -518.307,E2 -518.307} C_VEL
LIN {X 0,Y 608.409,Z 269.379,A -85,B 0,C 180,E1 -519.512,E2 -519.512} C_VEL
LIN {X 0,Y 608.671,Z 273.442,A -85,B 0,C 180,E1 -519.586,E2 -519.586} C_VEL
LIN {X 0,Y 608.655,Z 288.814,A -85,B 0,C 180,E1 -519.887,E2 -519.887} C_VEL
LIN {X 0,Y 608.656,Z 303.324,A -85,B 0,C 180,E1 -520.305,E2 -520.305} C_VEL
LIN {X 0,Y 608.585,Z 318.174,A -85,B 0,C 180,E1 -520.872,E2 -520.872} C_VEL
LIN {X 0,Y 608.581,Z 331.28,A -85,B 0,C 180,E1 -521.508,E2 -521.508} C_VEL
LIN {X 0,Y 608.542,Z 344.128,A -85,B 0,C 180,E1 -522.266,E2 -522.266} C_VEL
LIN {X 0,Y 608.532,Z 356.316,A -85,B 0,C 180,E1 -523.132,E2 -523.132} C_VEL
LIN {X 0,Y 608.503,Z 367.55,A -85,B 0,C 180,E1 -524.08,E2 -524.08} C_VEL
LIN {X 0,Y 608.486,Z 377.851,A -85,B 0,C 180,E1 -525.109,E2 -525.109} C_VEL
LIN {X 0,Y 608.473,Z 387.879,A -85,B 0,C 180,E1 -526.304,E2 -526.304} C_VEL
LIN {X 0,Y 608.464,Z 396.203,A -85,B 0,C 180,E1 -527.493,E2 -527.493} C_VEL
LIN {X 0,Y 608.458,Z 403.049,A -85,B 0,C 180,E1 -528.676,E2 -528.676} C_VEL
LIN {X 0,Y 608.437,Z 409.371,A -85,B 0,C 180,E1 -530.023,E2 -530.023} C_VEL
LIN {X 0,Y 608.423,Z 414.245,A -85,B 0,C 180,E1 -531.364,E2 -531.364} C_VEL
LIN {X 0,Y 608.423,Z 417.813,A -85,B 0,C 180,E1 -532.7,E2 -532.7} C_VEL
LIN {X 0,Y 608.435,Z 420.161,A -85,B 0,C 180,E1 -534.033,E2 -534.033} C_VEL
LIN {X 0,Y 608.43,Z 421.344,A -85,B 0,C 180,E1 -535.362,E2 -535.362} C_VEL
LIN {X 0,Y 608.416,Z 421.355,A -85,B 0,C 180,E1 -536.689,E2 -536.689} C_VEL
LIN {X 0,Y 608.445,Z 420.211,A -85,B 0,C 180,E1 -538.014,E2 -538.014} C_VEL
LIN {X 0,Y 608.435,Z 417.924,A -85,B 0,C 180,E1 -539.338,E2 -539.338} C_VEL
LIN {X 0,Y 608.434,Z 414.449,A -85,B 0,C 180,E1 -540.662,E2 -540.662} C_VEL
LIN {X 0,Y 608.445,Z 409.72,A -85,B 0,C 180,E1 -541.986,E2 -541.986} C_VEL
LIN {X 0,Y 608.433,Z 403.608,A -85,B 0,C 180,E1 -543.311,E2 -543.311} C_VEL
LIN {X 0,Y 608.462,Z 395.943,A -85,B 0,C 180,E1 -544.638,E2 -544.638} C_VEL
LIN {X 0,Y 608.477,Z 387.773,A -85,B 0,C 180,E1 -545.801,E2 -545.801} C_VEL
LIN {X 0,Y 608.49,Z 377.986,A -85,B 0,C 180,E1 -546.966,E2 -546.966} C_VEL
LIN {X 0,Y 608.491,Z 368.008,A -85,B 0,C 180,E1 -547.967,E2 -547.967} C_VEL
LIN {X 0,Y 608.527,Z 359.446,A -85,B 0,C 180,E1 -548.708,E2 -548.708} C_VEL
LIN {X 0,Y 607.933,Z 355.043,A -85,B 0,C 180,E1 -549.071,E2 -549.071} C_VEL
LIN {X 0,Y 605.145,Z 347.83,A -85,B 0,C 180,E1 -549.663,E2 -549.663} C_VEL
LIN {X 0,Y 602.323,Z 340.351,A -85,B 0,C 180,E1 -550.22,E2 -550.22} C_VEL
LIN {X 0,Y 601.669,Z 335.425,A -85,B 0,C 180,E1 -550.524,E2 -550.524} C_VEL
LIN {X 0,Y 601.69,Z 322.242,A -85,B 0,C 180,E1 -551.213,E2 -551.213} C_VEL
LIN {X 0,Y 601.763,Z 308.367,A -85,B 0,C 180,E1 -551.794,E2 -551.794} C_VEL
LIN {X 0,Y 601.849,Z 293.034,A -85,B 0,C 180,E1 -552.284,E2 -552.284} C_VEL
LIN {X 0,Y 601.871,Z 277.738,A -85,B 0,C 180,E1 -552.626,E2 -552.626} C_VEL
LIN {X 0,Y 601.644,Z 271.313,A -85,B 0,C 180,E1 -552.732,E2 -552.732} C_VEL
LIN {X 0,Y 601.324,Z 269.368,A -85,B 0,C 180,E1 -552.788,E2 -552.788} C_VEL
LIN {X 0,Y 601.297,Z 266.728,A -85,B 0,C 180,E1 -554.9,E2 -554.9} C_VEL
LIN {X 0,Y 601.323,Z 264.148,A -85,B 0,C 180,E1 -556.989,E2 -556.989} C_VEL
LIN {X 0,Y 601.311,Z 260.721,A -85,B 0,C 180,E1 -559.813,E2 -559.813} C_VEL
LIN {X 0,Y 601.317,Z 257.431,A -85,B 0,C 180,E1 -562.582,E2 -562.582} C_VEL
LIN {X 0,Y 601.333,Z 254.756,A -85,B 0,C 180,E1 -564.882,E2 -564.882} C_VEL
LIN {X 0,Y 601.337,Z 252.05,A -85,B 0,C 180,E1 -567.347,E2 -567.347} C_VEL
LIN {X 0,Y 601.343,Z 249.015,A -85,B 0,C 180,E1 -570.169,E2 -570.169} C_VEL
LIN {X 0,Y 601.363,Z 246.304,A -85,B 0,C 180,E1 -572.706,E2 -572.706} C_VEL
LIN {X 0,Y 601.372,Z 245.204,A -85,B 0,C 180,E1 -574.122,E2 -574.122} C_VEL
LIN {X 0,Y 601.397,Z 245.196,A -85,B 0,C 180,E1 -576.584,E2 -576.584} C_VEL
LIN {X 0,Y 601.418,Z 245.193,A -85,B 0,C 180,E1 -579.533,E2 -579.533} C_VEL
LIN {X 0,Y 601.417,Z 245.198,A -85,B 0,C 180,E1 -581.766,E2 -581.766} C_VEL
LIN {X 0,Y 601.402,Z 245.199,A -85,B 0,C 180,E1 -584.532,E2 -584.532} C_VEL
LIN {X 0,Y 601.418,Z 245.195,A -85,B 0,C 180,E1 -587.409,E2 -587.409} C_VEL
LIN {X 0,Y 601.382,Z 245.198,A -85,B 0,C 180,E1 -590.002,E2 -590.002} C_VEL
LIN {X 0,Y 601.439,Z 245.193,A -85,B 0,C 180,E1 -592.618,E2 -592.618} C_VEL
LIN {X 0,Y 601.417,Z 245.196,A -85,B 0,C 180,E1 -595.068,E2 -595.068} C_VEL
LIN {X 0,Y 601.401,Z 245.195,A -85,B 0,C 180,E1 -597.482,E2 -597.482} C_VEL
LIN {X 0,Y 601.433,Z 245.197,A -85,B 0,C 180,E1 -599.851,E2 -599.851} C_VEL
LIN {X 0,Y 601.421,Z 245.195,A -85,B 0,C 180,E1 -602.637,E2 -602.637} C_VEL
LIN {X 0,Y 601.39,Z 245.197,A -85,B 0,C 180,E1 -605.121,E2 -605.121} C_VEL
LIN {X 0,Y 601.42,Z 245.194,A -85,B 0,C 180,E1 -608.041,E2 -608.041} C_VEL
LIN {X 0,Y 601.41,Z 245.196,A -85,B 0,C 180,E1 -610.901,E2 -610.901} C_VEL
LIN {X 0,Y 601.443,Z 245.195,A -85,B 0,C 180,E1 -613.713,E2 -613.713} C_VEL
LIN {X 0,Y 601.414,Z 245.197,A -85,B 0,C 180,E1 -616.484,E2 -616.484} C_VEL
LIN {X 0,Y 601.388,Z 245.198,A -85,B 0,C 180,E1 -619.223,E2 -619.223} C_VEL
LIN {X 0,Y 601.443,Z 245.19,A -85,B 0,C 180,E1 -621.939,E2 -621.939} C_VEL
LIN {X 0,Y 601.407,Z 245.196,A -85,B 0,C 180,E1 -624.636,E2 -624.636} C_VEL
LIN {X 0,Y 601.445,Z 245.196,A -85,B 0,C 180,E1 -627.321,E2 -627.321} C_VEL
LIN {X 0,Y 601.449,Z 245.191,A -85,B 0,C 180,E1 -630,E2 -630} C_VEL
LIN {X 0,Y 601.415,Z 245.193,A -85,B 0,C 180,E1 -632.679,E2 -632.679} C_VEL
LIN {X 0,Y 601.428,Z 245.193,A -85,B 0,C 180,E1 -635.364,E2 -635.364} C_VEL
LIN {X 0,Y 601.437,Z 245.196,A -85,B 0,C 180,E1 -638.061,E2 -638.061} C_VEL
LIN {X 0,Y 601.421,Z 245.199,A -85,B 0,C 180,E1 -641.008,E2 -641.008} C_VEL
LIN {X 0,Y 601.414,Z 245.194,A -85,B 0,C 180,E1 -643.516,E2 -643.516} C_VEL
LIN {X 0,Y 601.406,Z 245.195,A -85,B 0,C 180,E1 -646.614,E2 -646.614} C_VEL
LIN {X 0,Y 601.422,Z 245.194,A -85,B 0,C 180,E1 -649.099,E2 -649.099} C_VEL
LIN {X 0,Y 601.396,Z 245.199,A -85,B 0,C 180,E1 -651.96,E2 -651.96} C_VEL
LIN {X 0,Y 601.4,Z 245.2,A -85,B 0,C 180,E1 -654.879,E2 -654.879} C_VEL
LIN {X 0,Y 601.413,Z 245.195,A -85,B 0,C 180,E1 -657.361,E2 -657.361} C_VEL
LIN {X 0,Y 601.402,Z 245.195,A -85,B 0,C 180,E1 -660.166,E2 -660.166} C_VEL
LIN {X 0,Y 601.428,Z 245.194,A -85,B 0,C 180,E1 -662.716,E2 -662.716} C_VEL
LIN {X 0,Y 601.383,Z 245.2,A -85,B 0,C 180,E1 -665.11,E2 -665.11} C_VEL
LIN {X 0,Y 601.437,Z 245.192,A -85,B 0,C 180,E1 -667.419,E2 -667.419} C_VEL
LIN {X 0,Y 601.407,Z 245.201,A -85,B 0,C 180,E1 -669.996,E2 -669.996} C_VEL
LIN {X 0,Y 601.379,Z 245.2,A -85,B 0,C 180,E1 -672.674,E2 -672.674} C_VEL
LIN {X 0,Y 601.431,Z 245.192,A -85,B 0,C 180,E1 -675.482,E2 -675.482} C_VEL
LIN {X 0,Y 601.418,Z 245.193,A -85,B 0,C 180,E1 -678.408,E2 -678.408} C_VEL
LIN {X 0,Y 601.413,Z 245.194,A -85,B 0,C 180,E1 -681.532,E2 -681.532} C_VEL
LIN {X 0,Y 601.4,Z 245.201,A -85,B 0,C 180,E1 -683.74,E2 -683.74} C_VEL
LIN {X 0,Y 601.406,Z 245.195,A -85,B 0,C 180,E1 -686.069,E2 -686.069} C_VEL
LIN {X 0,Y 601.417,Z 245.193,A -85,B 0,C 180,E1 -689.058,E2 -689.058} C_VEL
LIN {X 0,Y 601.43,Z 245.197,A -85,B 0,C 180,E1 -691.373,E2 -691.373} C_VEL
LIN {X 0,Y 601.41,Z 245.198,A -85,B 0,C 180,E1 -694.134,E2 -694.134} C_VEL
LIN {X 0,Y 601.403,Z 245.195,A -85,B 0,C 180,E1 -696.589,E2 -696.589} C_VEL
LIN {X 0,Y 601.405,Z 245.195,A -85,B 0,C 180,E1 -699.477,E2 -699.477} C_VEL
LIN {X 0,Y 601.393,Z 245.198,A -85,B 0,C 180,E1 -702.311,E2 -702.311} C_VEL
LIN {X 0,Y 601.417,Z 245.194,A -85,B 0,C 180,E1 -704.409,E2 -704.409} C_VEL
LIN {X 0,Y 601.375,Z 245.198,A -85,B 0,C 180,E1 -707.171,E2 -707.171} C_VEL
LIN {X 0,Y 601.44,Z 245.192,A -85,B 0,C 180,E1 -709.905,E2 -709.905} C_VEL
LIN {X 0,Y 601.411,Z 245.2,A -85,B 0,C 180,E1 -712.614,E2 -712.614} C_VEL
LIN {X 0,Y 601.406,Z 245.197,A -85,B 0,C 180,E1 -715.308,E2 -715.308} C_VEL
LIN {X 0,Y 601.438,Z 245.191,A -85,B 0,C 180,E1 -717.991,E2 -717.991} C_VEL
LIN {X 0,Y 601.428,Z 245.193,A -85,B 0,C 180,E1 -720.669,E2 -720.669} C_VEL
LIN {X 0,Y 601.433,Z 245.197,A -85,B 0,C 180,E1 -723.349,E2 -723.349} C_VEL
LIN {X 0,Y 601.418,Z 245.196,A -85,B 0,C 180,E1 -726.037,E2 -726.037} C_VEL
LIN {X 0,Y 601.393,Z 245.196,A -85,B 0,C 180,E1 -728.738,E2 -728.738} C_VEL
LIN {X 0,Y 601.428,Z 245.192,A -85,B 0,C 180,E1 -731.458,E2 -731.458} C_VEL
LIN {X 0,Y 601.417,Z 245.196,A -85,B 0,C 180,E1 -734.205,E2 -734.205} C_VEL
LIN {X 0,Y 601.414,Z 245.2,A -85,B 0,C 180,E1 -736.986,E2 -736.986} C_VEL
LIN {X 0,Y 601.402,Z 245.199,A -85,B 0,C 180,E1 -739.809,E2 -739.809} C_VEL
LIN {X 0,Y 601.405,Z 245.196,A -85,B 0,C 180,E1 -742.683,E2 -742.683} C_VEL
LIN {X 0,Y 601.402,Z 245.198,A -85,B 0,C 180,E1 -744.878,E2 -744.878} C_VEL
LIN {X 0,Y 601.408,Z 245.197,A -85,B 0,C 180,E1 -747.36,E2 -747.36} C_VEL
LIN {X 0,Y 601.403,Z 245.196,A -85,B 0,C 180,E1 -750.165,E2 -750.165} C_VEL
LIN {X 0,Y 601.421,Z 245.194,A -85,B 0,C 180,E1 -752.714,E2 -752.714} C_VEL
LIN {X 0,Y 601.375,Z 245.203,A -85,B 0,C 180,E1 -755.108,E2 -755.108} C_VEL
LIN {X 0,Y 601.438,Z 245.191,A -85,B 0,C 180,E1 -757.419,E2 -757.419} C_VEL
LIN {X 0,Y 601.415,Z 245.197,A -85,B 0,C 180,E1 -759.995,E2 -759.995} C_VEL
LIN {X 0,Y 601.384,Z 245.201,A -85,B 0,C 180,E1 -762.673,E2 -762.673} C_VEL
LIN {X 0,Y 601.429,Z 245.194,A -85,B 0,C 180,E1 -765.482,E2 -765.482} C_VEL
LIN {X 0,Y 601.434,Z 245.306,A -85,B 0,C 180,E1 -768.179,E2 -768.179} C_VEL
LIN {X 0,Y 601.582,Z 248.681,A -85,B 0,C 180,E1 -769.408,E2 -769.408} C_VEL
LIN {X 0,Y 601.588,Z 256.592,A -85,B 0,C 180,E1 -772.169,E2 -772.169} C_VEL
LIN {X 0,Y 601.544,Z 265.256,A -85,B 0,C 180,E1 -775.076,E2 -775.076} C_VEL
LIN {X 0,Y 601.527,Z 272.683,A -85,B 0,C 180,E1 -777.49,E2 -777.49} C_VEL
LIN {X 0,Y 601.481,Z 281.348,A -85,B 0,C 180,E1 -780.225,E2 -780.225} C_VEL
LIN {X 0,Y 601.463,Z 290.013,A -85,B 0,C 180,E1 -782.889,E2 -782.889} C_VEL
LIN {X 0,Y 601.413,Z 299.426,A -85,B 0,C 180,E1 -785.712,E2 -785.712} C_VEL
LIN {X 0,Y 601.416,Z 308.58,A -85,B 0,C 180,E1 -788.401,E2 -788.401} C_VEL
LIN {X 0,Y 601.349,Z 318.299,A -85,B 0,C 180,E1 -791.2,E2 -791.2} C_VEL
LIN {X 0,Y 601.366,Z 325.4,A -85,B 0,C 180,E1 -793.218,E2 -793.218} C_VEL
LIN {X 0,Y 601.867,Z 328.99,A -85,B 0,C 180,E1 -793.285,E2 -793.285} C_VEL
LIN {X 0,Y 601.839,Z 344.945,A -85,B 0,C 180,E1 -793.562,E2 -793.562} C_VEL
LIN {X 0,Y 601.811,Z 359.293,A -85,B 0,C 180,E1 -793.941,E2 -793.941} C_VEL
LIN {X 0,Y 601.733,Z 373.791,A -85,B 0,C 180,E1 -794.46,E2 -794.46} C_VEL
LIN {X 0,Y 601.664,Z 387.861,A -85,B 0,C 180,E1 -795.109,E2 -795.109} C_VEL
LIN {X 0,Y 601.615,Z 401.584,A -85,B 0,C 180,E1 -795.894,E2 -795.894} C_VEL
LIN {X 0,Y 601.57,Z 415.011,A -85,B 0,C 180,E1 -796.831,E2 -796.831} C_VEL
LIN {X 0,Y 601.514,Z 427.189,A -85,B 0,C 180,E1 -797.859,E2 -797.859} C_VEL
LIN {X 0,Y 601.437,Z 438.276,A -85,B 0,C 180,E1 -798.982,E2 -798.982} C_VEL
LIN {X 0,Y 601.427,Z 447.366,A -85,B 0,C 180,E1 -800.075,E2 -800.075} C_VEL
LIN {X 0,Y 601.388,Z 455.656,A -85,B 0,C 180,E1 -801.262,E2 -801.262} C_VEL
LIN {X 0,Y 601.365,Z 463.428,A -85,B 0,C 180,E1 -802.614,E2 -802.614} C_VEL
LIN {X 0,Y 601.357,Z 469.609,A -85,B 0,C 180,E1 -803.962,E2 -803.962} C_VEL
LIN {X 0,Y 601.33,Z 474.384,A -85,B 0,C 180,E1 -805.307,E2 -805.307} C_VEL
LIN {X 0,Y 601.337,Z 477.886,A -85,B 0,C 180,E1 -806.65,E2 -806.65} C_VEL
LIN {X 0,Y 601.343,Z 480.191,A -85,B 0,C 180,E1 -807.991,E2 -807.991} C_VEL
LIN {X 0,Y 601.335,Z 481.351,A -85,B 0,C 180,E1 -809.33,E2 -809.33} C_VEL
LIN {X 0,Y 601.335,Z 481.351,A -85,B 0,C 180,E1 -810.67,E2 -810.67} C_VEL
LIN {X 0,Y 601.343,Z 480.191,A -85,B 0,C 180,E1 -812.009,E2 -812.009} C_VEL
LIN {X 0,Y 601.337,Z 477.886,A -85,B 0,C 180,E1 -813.35,E2 -813.35} C_VEL
LIN {X 0,Y 601.33,Z 474.384,A -85,B 0,C 180,E1 -814.693,E2 -814.693} C_VEL
LIN {X 0,Y 601.357,Z 469.609,A -85,B 0,C 180,E1 -816.038,E2 -816.038} C_VEL
LIN {X 0,Y 601.365,Z 463.428,A -85,B 0,C 180,E1 -817.386,E2 -817.386} C_VEL
LIN {X 0,Y 601.388,Z 455.656,A -85,B 0,C 180,E1 -818.738,E2 -818.738} C_VEL
LIN {X 0,Y 601.427,Z 447.367,A -85,B 0,C 180,E1 -819.925,E2 -819.925} C_VEL
LIN {X 0,Y 601.46,Z 436.936,A -85,B 0,C 180,E1 -821.165,E2 -821.165} C_VEL
LIN {X 0,Y 601.514,Z 427.191,A -85,B 0,C 180,E1 -822.141,E2 -822.141} C_VEL
LIN {X 0,Y 601.57,Z 415.011,A -85,B 0,C 180,E1 -823.168,E2 -823.168} C_VEL
LIN {X 0,Y 601.606,Z 403.083,A -85,B 0,C 180,E1 -824.012,E2 -824.012} C_VEL
LIN {X 0,Y 601.676,Z 389.534,A -85,B 0,C 180,E1 -824.804,E2 -824.804} C_VEL
LIN {X 0,Y 601.72,Z 374.841,A -85,B 0,C 180,E1 -825.496,E2 -825.496} C_VEL
LIN {X 0,Y 601.806,Z 360.622,A -85,B 0,C 180,E1 -826.016,E2 -826.016} C_VEL
LIN {X 0,Y 601.841,Z 345.808,A -85,B 0,C 180,E1 -826.418,E2 -826.418} C_VEL
LIN {X 0,Y 601.855,Z 330.529,A -85,B 0,C 180,E1 -826.693,E2 -826.693} C_VEL
LIN {X 0,Y 601.554,Z 326.707,A -85,B 0,C 180,E1 -826.753,E2 -826.753} C_VEL
LIN {X 0,Y 601.367,Z 325.395,A -85,B 0,C 180,E1 -826.783,E2 -826.783} C_VEL
LIN {X 0,Y 601.412,Z 316.007,A -85,B 0,C 180,E1 -829.454,E2 -829.454} C_VEL
LIN {X 0,Y 601.415,Z 306.243,A -85,B 0,C 180,E1 -832.28,E2 -832.28} C_VEL
LIN {X 0,Y 601.432,Z 297.44,A -85,B 0,C 180,E1 -834.877,E2 -834.877} C_VEL
LIN {X 0,Y 601.464,Z 289.156,A -85,B 0,C 180,E1 -837.371,E2 -837.371} C_VEL
LIN {X 0,Y 601.482,Z 281.348,A -85,B 0,C 180,E1 -839.775,E2 -839.775} C_VEL
LIN {X 0,Y 601.527,Z 272.684,A -85,B 0,C 180,E1 -842.51,E2 -842.51} C_VEL
LIN {X 0,Y 601.564,Z 264.613,A -85,B 0,C 180,E1 -845.135,E2 -845.135} C_VEL
LIN {X 0,Y 601.588,Z 256.592,A -85,B 0,C 180,E1 -847.831,E2 -847.831} C_VEL
LIN {X 0,Y 601.582,Z 248.681,A -85,B 0,C 180,E1 -850.592,E2 -850.592} C_VEL
LIN {X 0,Y 601.469,Z 245.745,A -85,B 0,C 180,E1 -851.762,E2 -851.762} C_VEL
LIN {X 0,Y 601.38,Z 245.202,A -85,B 0,C 180,E1 -852.22,E2 -852.22} C_VEL
LIN {X 0,Y 601.399,Z 245.201,A -85,B 0,C 180,E1 -854.533,E2 -854.533} C_VEL
LIN {X 0,Y 601.387,Z 245.198,A -85,B 0,C 180,E1 -857.328,E2 -857.328} C_VEL
LIN {X 0,Y 601.424,Z 245.745,A -85,B 0,C 180,E1 -858.407,E2 -858.407} C_VEL
LIN {X 0,Y 601.412,Z 248.627,A -85,B 0,C 180,E1 -860.874,E2 -860.874} C_VEL
LIN {X 0,Y 601.398,Z 251.388,A -85,B 0,C 180,E1 -863.74,E2 -863.74} C_VEL
LIN {X 0,Y 601.352,Z 254.151,A -85,B 0,C 180,E1 -866.682,E2 -866.682} C_VEL
LIN {X 0,Y 601.318,Z 256.896,A -85,B 0,C 180,E1 -869.052,E2 -869.052} C_VEL
LIN {X 0,Y 601.306,Z 259.631,A -85,B 0,C 180,E1 -871.367,E2 -871.367} C_VEL
LIN {X 0,Y 601.332,Z 262.986,A -85,B 0,C 180,E1 -874.15,E2 -874.15} C_VEL
LIN {X 0,Y 601.311,Z 265.978,A -85,B 0,C 180,E1 -876.585,E2 -876.585} C_VEL
LIN {X 0,Y 601.33,Z 269.387,A -85,B 0,C 180,E1 -879.318,E2 -879.318} C_VEL
LIN {X 0,Y 601.885,Z 273.12,A -85,B 0,C 180,E1 -879.391,E2 -879.391} C_VEL
LIN {X 0,Y 601.843,Z 288.616,A -85,B 0,C 180,E1 -879.694,E2 -879.694} C_VEL
LIN {X 0,Y 601.819,Z 303.166,A -85,B 0,C 180,E1 -880.116,E2 -880.116} C_VEL
LIN {X 0,Y 601.694,Z 318.061,A -85,B 0,C 180,E1 -880.689,E2 -880.689} C_VEL
LIN {X 0,Y 601.667,Z 332.28,A -85,B 0,C 180,E1 -881.393,E2 -881.393} C_VEL
LIN {X 0,Y 601.593,Z 346.007,A -85,B 0,C 180,E1 -882.23,E2 -882.23} C_VEL
LIN {X 0,Y 601.564,Z 358.18,A -85,B 0,C 180,E1 -883.131,E2 -883.131} C_VEL
LIN {X 0,Y 601.493,Z 368.853,A -85,B 0,C 180,E1 -884.063,E2 -884.063} C_VEL
LIN {X 0,Y 601.448,Z 378.936,A -85,B 0,C 180,E1 -885.104,E2 -885.104} C_VEL
LIN {X 0,Y 601.412,Z 387.955,A -85,B 0,C 180,E1 -886.198,E2 -886.198} C_VEL
LIN {X 0,Y 601.395,Z 396.945,A -85,B 0,C 180,E1 -887.515,E2 -887.515} C_VEL
LIN {X 0,Y 601.363,Z 404.522,A -85,B 0,C 180,E1 -888.878,E2 -888.878} C_VEL
LIN {X 0,Y 601.344,Z 410.553,A -85,B 0,C 180,E1 -890.244,E2 -890.244} C_VEL
LIN {X 0,Y 601.344,Z 414.098,A -85,B 0,C 180,E1 -891.261,E2 -891.261} C_VEL
LIN {X 0,Y 601.323,Z 417.712,A -85,B 0,C 180,E1 -892.614,E2 -892.614} C_VEL
LIN {X 0,Y 601.334,Z 420.108,A -85,B 0,C 180,E1 -893.962,E2 -893.962} C_VEL
LIN {X 0,Y 601.327,Z 421.324,A -85,B 0,C 180,E1 -895.307,E2 -895.307} C_VEL
LIN {X 0,Y 601.333,Z 421.366,A -85,B 0,C 180,E1 -896.65,E2 -896.65} C_VEL
LIN {X 0,Y 601.343,Z 420.268,A -85,B 0,C 180,E1 -897.991,E2 -897.991} C_VEL
LIN {X 0,Y 601.336,Z 418.025,A -85,B 0,C 180,E1 -899.331,E2 -899.331} C_VEL
LIN {X 0,Y 601.336,Z 414.598,A -85,B 0,C 180,E1 -900.67,E2 -900.67} C_VEL
LIN {X 0,Y 601.352,Z 409.92,A -85,B 0,C 180,E1 -902.009,E2 -902.009} C_VEL
LIN {X 0,Y 601.351,Z 403.847,A -85,B 0,C 180,E1 -903.35,E2 -903.35} C_VEL
LIN {X 0,Y 601.399,Z 396.24,A -85,B 0,C 180,E1 -904.692,E2 -904.692} C_VEL
LIN {X 0,Y 601.413,Z 388.122,A -85,B 0,C 180,E1 -905.869,E2 -905.869} C_VEL
LIN {X 0,Y 601.45,Z 378.402,A -85,B 0,C 180,E1 -907.048,E2 -907.048} C_VEL
LIN {X 0,Y 601.495,Z 368.503,A -85,B 0,C 180,E1 -908.06,E2 -908.06} C_VEL
LIN {X 0,Y 601.528,Z 356.765,A -85,B 0,C 180,E1 -909.075,E2 -909.075} C_VEL
LIN {X 0,Y 601.597,Z 343.811,A -85,B 0,C 180,E1 -910.007,E2 -910.007} C_VEL
LIN {X 0,Y 601.669,Z 335.425,A -85,B 0,C 180,E1 -910.524,E2 -910.524} C_VEL
LIN {X 0,Y 601.085,Z 330.391,A -85,B 0,C 180,E1 -910.817,E2 -910.817} C_VEL
LIN {X 0,Y 598.274,Z 322.299,A -85,B 0,C 180,E1 -911.299,E2 -911.299} C_VEL
LIN {X 0,Y 595.489,Z 314.003,A -85,B 0,C 180,E1 -911.742,E2 -911.742} C_VEL
LIN {X 0,Y 594.92,Z 308.657,A -85,B 0,C 180,E1 -911.968,E2 -911.968} C_VEL
LIN {X 0,Y 595.033,Z 293.962,A -85,B 0,C 180,E1 -912.448,E2 -912.448} C_VEL
LIN {X 0,Y 595.074,Z 279.129,A -85,B 0,C 180,E1 -912.794,E2 -912.794} C_VEL
LIN {X 0,Y 594.93,Z 272.891,A -85,B 0,C 180,E1 -912.903,E2 -912.903} C_VEL
LIN {X 0,Y 594.224,Z 269.377,A -85,B 0,C 180,E1 -912.986,E2 -912.986} C_VEL
LIN {X 0,Y 594.213,Z 266.791,A -85,B 0,C 180,E1 -915.082,E2 -915.082} C_VEL
LIN {X 0,Y 594.229,Z 264.212,A -85,B 0,C 180,E1 -917.198,E2 -917.198} C_VEL
LIN {X 0,Y 594.202,Z 261.642,A -85,B 0,C 180,E1 -919.34,E2 -919.34} C_VEL
LIN {X 0,Y 594.213,Z 259.078,A -85,B 0,C 180,E1 -921.509,E2 -921.509} C_VEL
LIN {X 0,Y 594.276,Z 255.672,A -85,B 0,C 180,E1 -924.451,E2 -924.451} C_VEL
LIN {X 0,Y 594.253,Z 253.286,A -85,B 0,C 180,E1 -926.706,E2 -926.706} C_VEL
LIN {X 0,Y 594.246,Z 250.81,A -85,B 0,C 180,E1 -929.006,E2 -929.006} C_VEL
LIN {X 0,Y 594.302,Z 248.034,A -85,B 0,C 180,E1 -931.63,E2 -931.63} C_VEL
LIN {X 0,Y 594.297,Z 246.616,A -85,B 0,C 180,E1 -932.955,E2 -932.955} C_VEL
LIN {X 0,Y 594.327,Z 246.082,A -85,B 0,C 180,E1 -934.13,E2 -934.13} C_VEL
LIN {X 0,Y 594.382,Z 246.076,A -85,B 0,C 180,E1 -937.087,E2 -937.087} C_VEL
LIN {X 0,Y 594.362,Z 246.074,A -85,B 0,C 180,E1 -939.772,E2 -939.772} C_VEL
LIN {X 0,Y 594.347,Z 246.074,A -85,B 0,C 180,E1 -942.378,E2 -942.378} C_VEL
LIN {X 0,Y 594.34,Z 246.076,A -85,B 0,C 180,E1 -945.194,E2 -945.194} C_VEL
LIN {X 0,Y 594.373,Z 246.075,A -85,B 0,C 180,E1 -947.625,E2 -947.625} C_VEL
LIN {X 0,Y 594.359,Z 246.073,A -85,B 0,C 180,E1 -950.318,E2 -950.318} C_VEL
LIN {X 0,Y 594.385,Z 246.07,A -85,B 0,C 180,E1 -952.913,E2 -952.913} C_VEL
LIN {X 0,Y 594.375,Z 246.071,A -85,B 0,C 180,E1 -955.863,E2 -955.863} C_VEL
LIN {X 0,Y 594.37,Z 246.074,A -85,B 0,C 180,E1 -958.649,E2 -958.649} C_VEL
LIN {X 0,Y 594.387,Z 246.071,A -85,B 0,C 180,E1 -961.042,E2 -961.042} C_VEL
LIN {X 0,Y 594.381,Z 246.072,A -85,B 0,C 180,E1 -963.3,E2 -963.3} C_VEL
LIN {X 0,Y 594.37,Z 246.074,A -85,B 0,C 180,E1 -966.295,E2 -966.295} C_VEL
LIN {X 0,Y 594.396,Z 246.072,A -85,B 0,C 180,E1 -969.224,E2 -969.224} C_VEL
LIN {X 0,Y 594.338,Z 246.081,A -85,B 0,C 180,E1 -972.094,E2 -972.094} C_VEL
LIN {X 0,Y 594.369,Z 246.072,A -85,B 0,C 180,E1 -974.219,E2 -974.219} C_VEL
LIN {X 0,Y 594.381,Z 246.072,A -85,B 0,C 180,E1 -976.321,E2 -976.321} C_VEL
LIN {X 0,Y 594.349,Z 246.074,A -85,B 0,C 180,E1 -979.094,E2 -979.094} C_VEL
LIN {X 0,Y 594.416,Z 246.066,A -85,B 0,C 180,E1 -981.843,E2 -981.843} C_VEL
LIN {X 0,Y 594.375,Z 246.073,A -85,B 0,C 180,E1 -984.572,E2 -984.572} C_VEL
LIN {X 0,Y 594.41,Z 246.072,A -85,B 0,C 180,E1 -987.289,E2 -987.289} C_VEL
LIN {X 0,Y 594.418,Z 246.067,A -85,B 0,C 180,E1 -990,E2 -990} C_VEL
LIN {X 0,Y 594.385,Z 246.069,A -85,B 0,C 180,E1 -992.711,E2 -992.711} C_VEL
LIN {X 0,Y 594.394,Z 246.069,A -85,B 0,C 180,E1 -995.428,E2 -995.428} C_VEL
LIN {X 0,Y 594.38,Z 246.074,A -85,B 0,C 180,E1 -998.157,E2 -998.157} C_VEL
LIN {X 0,Y 594.385,Z 246.075,A -85,B 0,C 180,E1 -1001.07,E2 -1001.07} C_VEL
LIN {X 0,Y 594.38,Z 246.071,A -85,B 0,C 180,E1 -1003.679,E2 -1003.679} C_VEL
LIN {X 0,Y 594.36,Z 246.074,A -85,B 0,C 180,E1 -1006.707,E2 -1006.707} C_VEL
LIN {X 0,Y 594.371,Z 246.071,A -85,B 0,C 180,E1 -1009.334,E2 -1009.334} C_VEL
LIN {X 0,Y 594.357,Z 246.076,A -85,B 0,C 180,E1 -1011.504,E2 -1011.504} C_VEL
LIN {X 0,Y 594.392,Z 246.071,A -85,B 0,C 180,E1 -1014.446,E2 -1014.446} C_VEL
LIN {X 0,Y 594.381,Z 246.071,A -85,B 0,C 180,E1 -1016.7,E2 -1016.7} C_VEL
LIN {X 0,Y 594.372,Z 246.073,A -85,B 0,C 180,E1 -1018.999,E2 -1018.999} C_VEL
LIN {X 0,Y 594.381,Z 246.07,A -85,B 0,C 180,E1 -1021.643,E2 -1021.643} C_VEL
LIN {X 0,Y 594.372,Z 246.071,A -85,B 0,C 180,E1 -1024.581,E2 -1024.581} C_VEL
LIN {X 0,Y 594.39,Z 246.069,A -85,B 0,C 180,E1 -1027.608,E2 -1027.608} C_VEL
LIN {X 0,Y 594.37,Z 246.072,A -85,B 0,C 180,E1 -1030.567,E2 -1030.567} C_VEL
LIN {X 0,Y 594.346,Z 246.076,A -85,B 0,C 180,E1 -1033.302,E2 -1033.302} C_VEL
LIN {X 0,Y 594.373,Z 246.076,A -85,B 0,C 180,E1 -1036.161,E2 -1036.161} C_VEL
LIN {X 0,Y 594.377,Z 246.071,A -85,B 0,C 180,E1 -1038.535,E2 -1038.535} C_VEL
LIN {X 0,Y 594.374,Z 246.071,A -85,B 0,C 180,E1 -1041.298,E2 -1041.298} C_VEL
LIN {X 0,Y 594.354,Z 246.078,A -85,B 0,C 180,E1 -1043.755,E2 -1043.755} C_VEL
LIN {X 0,Y 594.356,Z 246.074,A -85,B 0,C 180,E1 -1046.237,E2 -1046.237} C_VEL
LIN {X 0,Y 594.373,Z 246.072,A -85,B 0,C 180,E1 -1048.65,E2 -1048.65} C_VEL
LIN {X 0,Y 594.387,Z 246.072,A -85,B 0,C 180,E1 -1051.042,E2 -1051.042} C_VEL
LIN {X 0,Y 594.37,Z 246.072,A -85,B 0,C 180,E1 -1053.3,E2 -1053.3} C_VEL
LIN {X 0,Y 594.404,Z 246.069,A -85,B 0,C 180,E1 -1055.564,E2 -1055.564} C_VEL
LIN {X 0,Y 594.366,Z 246.073,A -85,B 0,C 180,E1 -1058.496,E2 -1058.496} C_VEL
LIN {X 0,Y 594.359,Z 246.073,A -85,B 0,C 180,E1 -1061.382,E2 -1061.382} C_VEL
LIN {X 0,Y 594.37,Z 246.071,A -85,B 0,C 180,E1 -1064.219,E2 -1064.219} C_VEL
LIN {X 0,Y 594.366,Z 246.075,A -85,B 0,C 180,E1 -1066.321,E2 -1066.321} C_VEL
LIN {X 0,Y 594.373,Z 246.072,A -85,B 0,C 180,E1 -1069.094,E2 -1069.094} C_VEL
LIN {X 0,Y 594.386,Z 246.069,A -85,B 0,C 180,E1 -1071.843,E2 -1071.843} C_VEL
LIN {X 0,Y 594.369,Z 246.072,A -85,B 0,C 180,E1 -1074.572,E2 -1074.572} C_VEL
LIN {X 0,Y 594.406,Z 246.071,A -85,B 0,C 180,E1 -1077.289,E2 -1077.289} C_VEL
LIN {X 0,Y 594.418,Z 246.068,A -85,B 0,C 180,E1 -1080,E2 -1080} C_VEL
LIN {X 0,Y 594.393,Z 246.069,A -85,B 0,C 180,E1 -1082.711,E2 -1082.711} C_VEL
LIN {X 0,Y 594.388,Z 246.069,A -85,B 0,C 180,E1 -1085.428,E2 -1085.428} C_VEL
LIN {X 0,Y 594.36,Z 246.074,A -85,B 0,C 180,E1 -1088.157,E2 -1088.157} C_VEL
LIN {X 0,Y 594.392,Z 246.072,A -85,B 0,C 180,E1 -1091.072,E2 -1091.072} C_VEL
LIN {X 0,Y 594.378,Z 246.073,A -85,B 0,C 180,E1 -1093.679,E2 -1093.679} C_VEL
LIN {X 0,Y 594.367,Z 246.074,A -85,B 0,C 180,E1 -1096.709,E2 -1096.709} C_VEL
LIN {X 0,Y 594.369,Z 246.071,A -85,B 0,C 180,E1 -1099.334,E2 -1099.334} C_VEL
LIN {X 0,Y 594.354,Z 246.079,A -85,B 0,C 180,E1 -1101.504,E2 -1101.504} C_VEL
LIN {X 0,Y 594.393,Z 246.073,A -85,B 0,C 180,E1 -1104.446,E2 -1104.446} C_VEL
LIN {X 0,Y 594.379,Z 246.074,A -85,B 0,C 180,E1 -1107.461,E2 -1107.461} C_VEL
LIN {X 0,Y 594.369,Z 246.073,A -85,B 0,C 180,E1 -1110.324,E2 -1110.324} C_VEL
LIN {X 0,Y 594.38,Z 246.07,A -85,B 0,C 180,E1 -1112.95,E2 -1112.95} C_VEL
LIN {X 0,Y 594.321,Z 246.081,A -85,B 0,C 180,E1 -1115.411,E2 -1115.411} C_VEL
LIN {X 0,Y 594.387,Z 246.071,A -85,B 0,C 180,E1 -1117.941,E2 -1117.941} C_VEL
LIN {X 0,Y 594.375,Z 246.071,A -85,B 0,C 180,E1 -1120.821,E2 -1120.821} C_VEL
LIN {X 0,Y 594.354,Z 246.075,A -85,B 0,C 180,E1 -1123.838,E2 -1123.838} C_VEL
LIN {X 0,Y 594.368,Z 246.073,A -85,B 0,C 180,E1 -1126.7,E2 -1126.7} C_VEL
LIN {X 0,Y 594.369,Z 246.108,A -85,B 0,C 180,E1 -1127.843,E2 -1127.843} C_VEL
LIN {X 0,Y 594.691,Z 249.527,A -85,B 0,C 180,E1 -1129.143,E2 -1129.143} C_VEL
LIN {X 0,Y 594.651,Z 257.83,A -85,B 0,C 180,E1 -1132.079,E2 -1132.079} C_VEL
LIN {X 0,Y 594.606,Z 265.357,A -85,B 0,C 180,E1 -1134.642,E2 -1134.642} C_VEL
LIN {X 0,Y 594.565,Z 273.921,A -85,B 0,C 180,E1 -1137.464,E2 -1137.464} C_VEL
LIN {X 0,Y 594.503,Z 282.586,A -85,B 0,C 180,E1 -1140.23,E2 -1140.23} C_VEL
LIN {X 0,Y 594.455,Z 291.251,A -85,B 0,C 180,E1 -1142.924,E2 -1142.924} C_VEL
LIN {X 0,Y 594.398,Z 299.949,A -85,B 0,C 180,E1 -1145.564,E2 -1145.564} C_VEL
LIN {X 0,Y 594.38,Z 308.58,A -85,B 0,C 180,E1 -1148.132,E2 -1148.132} C_VEL
LIN {X 0,Y 594.362,Z 317.245,A -85,B 0,C 180,E1 -1150.665,E2 -1150.665} C_VEL
LIN {X 0,Y 594.307,Z 325.418,A -85,B 0,C 180,E1 -1153.018,E2 -1153.018} C_VEL
LIN {X 0,Y 595.059,Z 329.89,A -85,B 0,C 180,E1 -1153.102,E2 -1153.102} C_VEL
LIN {X 0,Y 595.037,Z 345.269,A -85,B 0,C 180,E1 -1153.376,E2 -1153.376} C_VEL
LIN {X 0,Y 594.969,Z 360.617,A -85,B 0,C 180,E1 -1153.795,E2 -1153.795} C_VEL
LIN {X 0,Y 594.864,Z 374.836,A -85,B 0,C 180,E1 -1154.32,E2 -1154.32} C_VEL
LIN {X 0,Y 594.761,Z 389.528,A -85,B 0,C 180,E1 -1155.02,E2 -1155.02} C_VEL
LIN {X 0,Y 594.673,Z 403.076,A -85,B 0,C 180,E1 -1155.822,E2 -1155.822} C_VEL
LIN {X 0,Y 594.596,Z 416.108,A -85,B 0,C 180,E1 -1156.761,E2 -1156.761} C_VEL
LIN {X 0,Y 594.53,Z 427.186,A -85,B 0,C 180,E1 -1157.715,E2 -1157.715} C_VEL
LIN {X 0,Y 594.455,Z 437.281,A -85,B 0,C 180,E1 -1158.739,E2 -1158.739} C_VEL
LIN {X 0,Y 594.387,Z 447.364,A -85,B 0,C 180,E1 -1159.956,E2 -1159.956} C_VEL
LIN {X 0,Y 594.331,Z 455.658,A -85,B 0,C 180,E1 -1161.157,E2 -1161.157} C_VEL
LIN {X 0,Y 594.287,Z 463.43,A -85,B 0,C 180,E1 -1162.525,E2 -1162.525} C_VEL
LIN {X 0,Y 594.279,Z 469.611,A -85,B 0,C 180,E1 -1163.89,E2 -1163.89} C_VEL
LIN {X 0,Y 594.232,Z 474.385,A -85,B 0,C 180,E1 -1165.251,E2 -1165.251} C_VEL
LIN {X 0,Y 594.257,Z 477.887,A -85,B 0,C 180,E1 -1166.61,E2 -1166.61} C_VEL
LIN {X 0,Y 594.241,Z 480.192,A -85,B 0,C 180,E1 -1167.967,E2 -1167.967} C_VEL
LIN {X 0,Y 594.235,Z 481.351,A -85,B 0,C 180,E1 -1169.322,E2 -1169.322} C_VEL
LIN {X 0,Y 594.235,Z 481.35,A -85,B 0,C 180,E1 -1170.678,E2 -1170.678} C_VEL
LIN {X 0,Y 594.241,Z 480.191,A -85,B 0,C 180,E1 -1172.033,E2 -1172.033} C_VEL
LIN {X 0,Y 594.257,Z 477.886,A -85,B 0,C 180,E1 -1173.39,E2 -1173.39} C_VEL
LIN {X 0,Y 594.232,Z 474.385,A -85,B 0,C 180,E1 -1174.749,E2 -1174.749} C_VEL
LIN {X 0,Y 594.279,Z 469.611,A -85,B 0,C 180,E1 -1176.11,E2 -1176.11} C_VEL
LIN {X 0,Y 594.287,Z 463.429,A -85,B 0,C 180,E1 -1177.475,E2 -1177.475} C_VEL
LIN {X 0,Y 594.331,Z 455.658,A -85,B 0,C 180,E1 -1178.843,E2 -1178.843} C_VEL
LIN {X 0,Y 594.387,Z 447.365,A -85,B 0,C 180,E1 -1180.044,E2 -1180.044} C_VEL
LIN {X 0,Y 594.433,Z 437.552,A -85,B 0,C 180,E1 -1181.231,E2 -1181.231} C_VEL
LIN {X 0,Y 594.53,Z 427.189,A -85,B 0,C 180,E1 -1182.285,E2 -1182.285} C_VEL
LIN {X 0,Y 594.581,Z 415.009,A -85,B 0,C 180,E1 -1183.326,E2 -1183.326} C_VEL
LIN {X 0,Y 594.694,Z 403.082,A -85,B 0,C 180,E1 -1184.178,E2 -1184.178} C_VEL
LIN {X 0,Y 594.761,Z 389.533,A -85,B 0,C 180,E1 -1184.98,E2 -1184.98} C_VEL
LIN {X 0,Y 594.866,Z 374.837,A -85,B 0,C 180,E1 -1185.68,E2 -1185.68} C_VEL
LIN {X 0,Y 594.987,Z 360.628,A -85,B 0,C 180,E1 -1186.204,E2 -1186.204} C_VEL
LIN {X 0,Y 595.039,Z 345.253,A -85,B 0,C 180,E1 -1186.624,E2 -1186.624} C_VEL
LIN {X 0,Y 595.082,Z 329.885,A -85,B 0,C 180,E1 -1186.898,E2 -1186.898} C_VEL
LIN {X 0,Y 594.307,Z 325.417,A -85,B 0,C 180,E1 -1186.983,E2 -1186.983} C_VEL
LIN {X 0,Y 594.358,Z 316.007,A -85,B 0,C 180,E1 -1189.694,E2 -1189.694} C_VEL
LIN {X 0,Y 594.368,Z 307.342,A -85,B 0,C 180,E1 -1192.233,E2 -1192.233} C_VEL
LIN {X 0,Y 594.414,Z 298.678,A -85,B 0,C 180,E1 -1194.818,E2 -1194.818} C_VEL
LIN {X 0,Y 594.461,Z 289.742,A -85,B 0,C 180,E1 -1197.541,E2 -1197.541} C_VEL
LIN {X 0,Y 594.521,Z 280.746,A -85,B 0,C 180,E1 -1200.35,E2 -1200.35} C_VEL
LIN {X 0,Y 594.563,Z 272.684,A -85,B 0,C 180,E1 -1202.939,E2 -1202.939} C_VEL
LIN {X 0,Y 594.606,Z 265.257,A -85,B 0,C 180,E1 -1205.392,E2 -1205.392} C_VEL
LIN {X 0,Y 594.651,Z 257.83,A -85,B 0,C 180,E1 -1207.921,E2 -1207.921} C_VEL
LIN {X 0,Y 594.657,Z 250.403,A -85,B 0,C 180,E1 -1210.544,E2 -1210.544} C_VEL
LIN {X 0,Y 594.613,Z 247.529,A -85,B 0,C 180,E1 -1211.873,E2 -1211.873} C_VEL
LIN {X 0,Y 594.341,Z 246.081,A -85,B 0,C 180,E1 -1212.85,E2 -1212.85} C_VEL
LIN {X 0,Y 594.361,Z 246.074,A -85,B 0,C 180,E1 -1215.762,E2 -1215.762} C_VEL
LIN {X 0,Y 594.349,Z 246.078,A -85,B 0,C 180,E1 -1217.623,E2 -1217.623} C_VEL
LIN {X 0,Y 594.377,Z 247.951,A -85,B 0,C 180,E1 -1219.434,E2 -1219.434} C_VEL
LIN {X 0,Y 594.323,Z 250.636,A -85,B 0,C 180,E1 -1222.055,E2 -1222.055} C_VEL
LIN {X 0,Y 594.305,Z 253.032,A -85,B 0,C 180,E1 -1224.683,E2 -1224.683} C_VEL
LIN {X 0,Y 594.255,Z 255.069,A -85,B 0,C 180,E1 -1227.108,E2 -1227.108} C_VEL
LIN {X 0,Y 594.244,Z 258.044,A -85,B 0,C 180,E1 -1229.696,E2 -1229.696} C_VEL
LIN {X 0,Y 594.265,Z 261.381,A -85,B 0,C 180,E1 -1232.534,E2 -1232.534} C_VEL
LIN {X 0,Y 594.246,Z 265.068,A -85,B 0,C 180,E1 -1235.598,E2 -1235.598} C_VEL
LIN {X 0,Y 594.215,Z 268.618,A -85,B 0,C 180,E1 -1238.491,E2 -1238.491} C_VEL
LIN {X 0,Y 594.246,Z 269.598,A -85,B 0,C 180,E1 -1239.118,E2 -1239.118} C_VEL
LIN {X 0,Y 595.079,Z 273.748,A -85,B 0,C 180,E1 -1239.204,E2 -1239.204} C_VEL
LIN {X 0,Y 595.041,Z 289.354,A -85,B 0,C 180,E1 -1239.519,E2 -1239.519} C_VEL
LIN {X 0,Y 594.958,Z 303.002,A -85,B 0,C 180,E1 -1239.922,E2 -1239.922} C_VEL
LIN {X 0,Y 594.806,Z 317.946,A -85,B 0,C 180,E1 -1240.501,E2 -1240.501} C_VEL
LIN {X 0,Y 594.738,Z 332.092,A -85,B 0,C 180,E1 -1241.208,E2 -1241.208} C_VEL
LIN {X 0,Y 594.649,Z 345.281,A -85,B 0,C 180,E1 -1242.015,E2 -1242.015} C_VEL
LIN {X 0,Y 594.596,Z 357.836,A -85,B 0,C 180,E1 -1242.949,E2 -1242.949} C_VEL
LIN {X 0,Y 594.496,Z 368.35,A -85,B 0,C 180,E1 -1243.87,E2 -1243.87} C_VEL
LIN {X 0,Y 594.412,Z 378.508,A -85,B 0,C 180,E1 -1244.923,E2 -1244.923} C_VEL
LIN {X 0,Y 594.362,Z 387.954,A -85,B 0,C 180,E1 -1246.08,E2 -1246.08} C_VEL
LIN {X 0,Y 594.343,Z 396.657,A -85,B 0,C 180,E1 -1247.364,E2 -1247.364} C_VEL
LIN {X 0,Y 594.306,Z 404.319,A -85,B 0,C 180,E1 -1248.749,E2 -1248.749} C_VEL
LIN {X 0,Y 594.262,Z 410.378,A -85,B 0,C 180,E1 -1250.126,E2 -1250.126} C_VEL
LIN {X 0,Y 594.245,Z 413.951,A -85,B 0,C 180,E1 -1251.156,E2 -1251.156} C_VEL
LIN {X 0,Y 594.249,Z 417.613,A -85,B 0,C 180,E1 -1252.525,E2 -1252.525} C_VEL
LIN {X 0,Y 594.239,Z 420.055,A -85,B 0,C 180,E1 -1253.89,E2 -1253.89} C_VEL
LIN {X 0,Y 594.225,Z 421.301,A -85,B 0,C 180,E1 -1255.251,E2 -1255.251} C_VEL
LIN {X 0,Y 594.253,Z 421.376,A -85,B 0,C 180,E1 -1256.61,E2 -1256.61} C_VEL
LIN {X 0,Y 594.241,Z 420.324,A -85,B 0,C 180,E1 -1257.967,E2 -1257.967} C_VEL
LIN {X 0,Y 594.237,Z 418.127,A -85,B 0,C 180,E1 -1259.323,E2 -1259.323} C_VEL
LIN {X 0,Y 594.239,Z 414.747,A -85,B 0,C 180,E1 -1260.678,E2 -1260.678} C_VEL
LIN {X 0,Y 594.258,Z 410.113,A -85,B 0,C 180,E1 -1262.033,E2 -1262.033} C_VEL
LIN {X 0,Y 594.273,Z 404.085,A -85,B 0,C 180,E1 -1263.39,E2 -1263.39} C_VEL
LIN {X 0,Y 594.339,Z 396.52,A -85,B 0,C 180,E1 -1264.748,E2 -1264.748} C_VEL
LIN {X 0,Y 594.35,Z 388.471,A -85,B 0,C 180,E1 -1265.939,E2 -1265.939} C_VEL
LIN {X 0,Y 594.413,Z 378.817,A -85,B 0,C 180,E1 -1267.132,E2 -1267.132} C_VEL
LIN {X 0,Y 594.524,Z 367.236,A -85,B 0,C 180,E1 -1268.326,E2 -1268.326} C_VEL
LIN {X 0,Y 594.597,Z 355.209,A -85,B 0,C 180,E1 -1269.353,E2 -1269.353} C_VEL
LIN {X 0,Y 594.691,Z 341.935,A -85,B 0,C 180,E1 -1270.297,E2 -1270.297} C_VEL
LIN {X 0,Y 594.768,Z 328.561,A -85,B 0,C 180,E1 -1271.076,E2 -1271.076} C_VEL
LIN {X 0,Y 594.86,Z 313.986,A -85,B 0,C 180,E1 -1271.759,E2 -1271.759} C_VEL
LIN {X 0,Y 594.92,Z 308.657,A -85,B 0,C 180,E1 -1271.968,E2 -1271.968} C_VEL
LIN {X 0,Y 594.437,Z 303.21,A -85,B 0,C 180,E1 -1272.183,E2 -1272.183} C_VEL
LIN {X 0,Y 591.701,Z 294.401,A -85,B 0,C 180,E1 -1272.538,E2 -1272.538} C_VEL
LIN {X 0,Y 588.893,Z 285.431,A -85,B 0,C 180,E1 -1272.844,E2 -1272.844} C_VEL
LIN {X 0,Y 588.287,Z 279.737,A -85,B 0,C 180,E1 -1272.981,E2 -1272.981} C_VEL
LIN {X 0,Y 588.117,Z 273.872,A -85,B 0,C 180,E1 -1273.089,E2 -1273.089} C_VEL
LIN {X 0,Y 587.126,Z 269.385,A -85,B 0,C 180,E1 -1273.19,E2 -1273.19} C_VEL
LIN {X 0,Y 587.148,Z 265.994,A -85,B 0,C 180,E1 -1275.98,E2 -1275.98} C_VEL
LIN {X 0,Y 587.137,Z 262.416,A -85,B 0,C 180,E1 -1278.98,E2 -1278.98} C_VEL
LIN {X 0,Y 587.131,Z 259.144,A -85,B 0,C 180,E1 -1281.782,E2 -1281.782} C_VEL
LIN {X 0,Y 587.177,Z 255.834,A -85,B 0,C 180,E1 -1284.767,E2 -1284.767} C_VEL
LIN {X 0,Y 587.167,Z 253.441,A -85,B 0,C 180,E1 -1287.055,E2 -1287.055} C_VEL
LIN {X 0,Y 587.182,Z 250.985,A -85,B 0,C 180,E1 -1289.389,E2 -1289.389} C_VEL
LIN {X 0,Y 587.224,Z 248.411,A -85,B 0,C 180,E1 -1291.816,E2 -1291.816} C_VEL
LIN {X 0,Y 587.227,Z 246.967,A -85,B 0,C 180,E1 -1293.404,E2 -1293.404} C_VEL
LIN {X 0,Y 587.289,Z 246.955,A -85,B 0,C 180,E1 -1295.9,E2 -1295.9} C_VEL
LIN {X 0,Y 587.321,Z 246.954,A -85,B 0,C 180,E1 -1298.48,E2 -1298.48} C_VEL
LIN {X 0,Y 587.34,Z 246.948,A -85,B 0,C 180,E1 -1301.157,E2 -1301.157} C_VEL
LIN {X 0,Y 587.307,Z 246.951,A -85,B 0,C 180,E1 -1304.111,E2 -1304.111} C_VEL
LIN {X 0,Y 587.319,Z 246.95,A -85,B 0,C 180,E1 -1306.994,E2 -1306.994} C_VEL
LIN {X 0,Y 587.305,Z 246.952,A -85,B 0,C 180,E1 -1309.745,E2 -1309.745} C_VEL
LIN {X 0,Y 587.344,Z 246.952,A -85,B 0,C 180,E1 -1312.392,E2 -1312.392} C_VEL
LIN {X 0,Y 587.345,Z 246.949,A -85,B 0,C 180,E1 -1315.653,E2 -1315.653} C_VEL
LIN {X 0,Y 587.335,Z 246.951,A -85,B 0,C 180,E1 -1318.23,E2 -1318.23} C_VEL
LIN {X 0,Y 587.354,Z 246.946,A -85,B 0,C 180,E1 -1320.867,E2 -1320.867} C_VEL
LIN {X 0,Y 587.331,Z 246.954,A -85,B 0,C 180,E1 -1322.954,E2 -1322.954} C_VEL
LIN {X 0,Y 587.342,Z 246.947,A -85,B 0,C 180,E1 -1325.423,E2 -1325.423} C_VEL
LIN {X 0,Y 587.327,Z 246.949,A -85,B 0,C 180,E1 -1328.226,E2 -1328.226} C_VEL
LIN {X 0,Y 587.331,Z 246.948,A -85,B 0,C 180,E1 -1331.15,E2 -1331.15} C_VEL
LIN {X 0,Y 587.325,Z 246.95,A -85,B 0,C 180,E1 -1334.025,E2 -1334.025} C_VEL
LIN {X 0,Y 587.36,Z 246.945,A -85,B 0,C 180,E1 -1336.154,E2 -1336.154} C_VEL
LIN {X 0,Y 587.341,Z 246.947,A -85,B 0,C 180,E1 -1338.962,E2 -1338.962} C_VEL
LIN {X 0,Y 587.368,Z 246.944,A -85,B 0,C 180,E1 -1341.745,E2 -1341.745} C_VEL
LIN {X 0,Y 587.343,Z 246.95,A -85,B 0,C 180,E1 -1344.507,E2 -1344.507} C_VEL
LIN {X 0,Y 587.375,Z 246.948,A -85,B 0,C 180,E1 -1347.257,E2 -1347.257} C_VEL
LIN {X 0,Y 587.387,Z 246.943,A -85,B 0,C 180,E1 -1350,E2 -1350} C_VEL
LIN {X 0,Y 587.354,Z 246.945,A -85,B 0,C 180,E1 -1352.743,E2 -1352.743} C_VEL
LIN {X 0,Y 587.36,Z 246.945,A -85,B 0,C 180,E1 -1355.493,E2 -1355.493} C_VEL
LIN {X 0,Y 587.339,Z 246.949,A -85,B 0,C 180,E1 -1358.256,E2 -1358.256} C_VEL
LIN {X 0,Y 587.353,Z 246.95,A -85,B 0,C 180,E1 -1361.134,E2 -1361.134} C_VEL
LIN {X 0,Y 587.359,Z 246.948,A -85,B 0,C 180,E1 -1363.846,E2 -1363.846} C_VEL
LIN {X 0,Y 587.332,Z 246.95,A -85,B 0,C 180,E1 -1366.807,E2 -1366.807} C_VEL
LIN {X 0,Y 587.316,Z 246.95,A -85,B 0,C 180,E1 -1369.576,E2 -1369.576} C_VEL
LIN {X 0,Y 587.312,Z 246.955,A -85,B 0,C 180,E1 -1371.775,E2 -1371.775} C_VEL
LIN {X 0,Y 587.354,Z 246.951,A -85,B 0,C 180,E1 -1374.759,E2 -1374.759} C_VEL
LIN {X 0,Y 587.344,Z 246.951,A -85,B 0,C 180,E1 -1377.691,E2 -1377.691} C_VEL
LIN {X 0,Y 587.323,Z 246.951,A -85,B 0,C 180,E1 -1380.507,E2 -1380.507} C_VEL
LIN {X 0,Y 587.345,Z 246.946,A -85,B 0,C 180,E1 -1383.112,E2 -1383.112} C_VEL
LIN {X 0,Y 587.278,Z 246.959,A -85,B 0,C 180,E1 -1385.534,E2 -1385.534} C_VEL
LIN {X 0,Y 587.338,Z 246.947,A -85,B 0,C 180,E1 -1387.838,E2 -1387.838} C_VEL
LIN {X 0,Y 587.316,Z 246.953,A -85,B 0,C 180,E1 -1390.255,E2 -1390.255} C_VEL
LIN {X 0,Y 587.293,Z 246.957,A -85,B 0,C 180,E1 -1393.116,E2 -1393.116} C_VEL
LIN {X 0,Y 587.328,Z 246.954,A -85,B 0,C 180,E1 -1396.05,E2 -1396.05} C_VEL
LIN {X 0,Y 587.336,Z 246.951,A -85,B 0,C 180,E1 -1398.926,E2 -1398.926} C_VEL
LIN {X 0,Y 587.324,Z 246.949,A -85,B 0,C 180,E1 -1401.52,E2 -1401.52} C_VEL
LIN {X 0,Y 587.295,Z 246.954,A -85,B 0,C 180,E1 -1404.1,E2 -1404.1} C_VEL
LIN {X 0,Y 587.336,Z 246.951,A -85,B 0,C 180,E1 -1406.89,E2 -1406.89} C_VEL
LIN {X 0,Y 587.338,Z 246.953,A -85,B 0,C 180,E1 -1409.83,E2 -1409.83} C_VEL
LIN {X 0,Y 587.346,Z 246.947,A -85,B 0,C 180,E1 -1412.309,E2 -1412.309} C_VEL
LIN {X 0,Y 587.359,Z 246.946,A -85,B 0,C 180,E1 -1415.42,E2 -1415.42} C_VEL
LIN {X 0,Y 587.323,Z 246.949,A -85,B 0,C 180,E1 -1418.226,E2 -1418.226} C_VEL
LIN {X 0,Y 587.332,Z 246.948,A -85,B 0,C 180,E1 -1421.15,E2 -1421.15} C_VEL
LIN {X 0,Y 587.325,Z 246.949,A -85,B 0,C 180,E1 -1424.025,E2 -1424.025} C_VEL
LIN {X 0,Y 587.347,Z 246.948,A -85,B 0,C 180,E1 -1426.154,E2 -1426.154} C_VEL
LIN {X 0,Y 587.343,Z 246.947,A -85,B 0,C 180,E1 -1428.962,E2 -1428.962} C_VEL
LIN {X 0,Y 587.346,Z 246.946,A -85,B 0,C 180,E1 -1431.744,E2 -1431.744} C_VEL
LIN {X 0,Y 587.337,Z 246.949,A -85,B 0,C 180,E1 -1434.507,E2 -1434.507} C_VEL
LIN {X 0,Y 587.372,Z 246.948,A -85,B 0,C 180,E1 -1437.257,E2 -1437.257} C_VEL
LIN {X 0,Y 587.387,Z 246.944,A -85,B 0,C 180,E1 -1440,E2 -1440} C_VEL
LIN {X 0,Y 587.362,Z 246.945,A -85,B 0,C 180,E1 -1442.743,E2 -1442.743} C_VEL
LIN {X 0,Y 587.354,Z 246.945,A -85,B 0,C 180,E1 -1445.493,E2 -1445.493} C_VEL
LIN {X 0,Y 587.325,Z 246.95,A -85,B 0,C 180,E1 -1448.256,E2 -1448.256} C_VEL
LIN {X 0,Y 587.354,Z 246.948,A -85,B 0,C 180,E1 -1451.133,E2 -1451.133} C_VEL
LIN {X 0,Y 587.345,Z 246.948,A -85,B 0,C 180,E1 -1454.25,E2 -1454.25} C_VEL
LIN {X 0,Y 587.347,Z 246.947,A -85,B 0,C 180,E1 -1457.406,E2 -1457.406} C_VEL
LIN {X 0,Y 587.313,Z 246.951,A -85,B 0,C 180,E1 -1459.576,E2 -1459.576} C_VEL
LIN {X 0,Y 587.311,Z 246.953,A -85,B 0,C 180,E1 -1461.775,E2 -1461.775} C_VEL
LIN {X 0,Y 587.355,Z 246.949,A -85,B 0,C 180,E1 -1464.758,E2 -1464.758} C_VEL
LIN {X 0,Y 587.304,Z 246.955,A -85,B 0,C 180,E1 -1467.82,E2 -1467.82} C_VEL
LIN {X 0,Y 587.324,Z 246.953,A -85,B 0,C 180,E1 -1470.507,E2 -1470.507} C_VEL
LIN {X 0,Y 587.341,Z 246.947,A -85,B 0,C 180,E1 -1473.111,E2 -1473.111} C_VEL
LIN {X 0,Y 587.272,Z 246.958,A -85,B 0,C 180,E1 -1475.533,E2 -1475.533} C_VEL
LIN {X 0,Y 587.342,Z 246.947,A -85,B 0,C 180,E1 -1477.838,E2 -1477.838} C_VEL
LIN {X 0,Y 587.316,Z 246.951,A -85,B 0,C 180,E1 -1480.254,E2 -1480.254} C_VEL
LIN {X 0,Y 587.295,Z 246.957,A -85,B 0,C 180,E1 -1483.116,E2 -1483.116} C_VEL
LIN {X 0,Y 587.326,Z 246.953,A -85,B 0,C 180,E1 -1486.049,E2 -1486.049} C_VEL
LIN {X 0,Y 587.358,Z 247.153,A -85,B 0,C 180,E1 -1487.592,E2 -1487.592} C_VEL
LIN {X 0,Y 587.784,Z 250.438,A -85,B 0,C 180,E1 -1488.881,E2 -1488.881} C_VEL
LIN {X 0,Y 587.708,Z 257.83,A -85,B 0,C 180,E1 -1491.55,E2 -1491.55} C_VEL
LIN {X 0,Y 587.667,Z 266.095,A -85,B 0,C 180,E1 -1494.412,E2 -1494.412} C_VEL
LIN {X 0,Y 587.597,Z 273.378,A -85,B 0,C 180,E1 -1496.85,E2 -1496.85} C_VEL
LIN {X 0,Y 587.507,Z 282.586,A -85,B 0,C 180,E1 -1499.839,E2 -1499.839} C_VEL
LIN {X 0,Y 587.469,Z 290.323,A -85,B 0,C 180,E1 -1502.285,E2 -1502.285} C_VEL
LIN {X 0,Y 587.409,Z 298.678,A -85,B 0,C 180,E1 -1504.866,E2 -1504.866} C_VEL
LIN {X 0,Y 587.342,Z 307.342,A -85,B 0,C 180,E1 -1507.486,E2 -1507.486} C_VEL
LIN {X 0,Y 587.305,Z 316.007,A -85,B 0,C 180,E1 -1510.059,E2 -1510.059} C_VEL
LIN {X 0,Y 587.255,Z 325.48,A -85,B 0,C 180,E1 -1512.812,E2 -1512.812} C_VEL
LIN {X 0,Y 588.266,Z 331.075,A -85,B 0,C 180,E1 -1512.918,E2 -1512.918} C_VEL
LIN {X 0,Y 588.239,Z 346.565,A -85,B 0,C 180,E1 -1513.21,E2 -1513.21} C_VEL
LIN {X 0,Y 588.134,Z 361.914,A -85,B 0,C 180,E1 -1513.646,E2 -1513.646} C_VEL
LIN {X 0,Y 587.998,Z 374.833,A -85,B 0,C 180,E1 -1514.132,E2 -1514.132} C_VEL
LIN {X 0,Y 587.864,Z 389.525,A -85,B 0,C 180,E1 -1514.84,E2 -1514.84} C_VEL
LIN {X 0,Y 587.757,Z 402.16,A -85,B 0,C 180,E1 -1515.59,E2 -1515.59} C_VEL
LIN {X 0,Y 587.629,Z 415.008,A -85,B 0,C 180,E1 -1516.513,E2 -1516.513} C_VEL
LIN {X 0,Y 587.521,Z 427.184,A -85,B 0,C 180,E1 -1517.566,E2 -1517.566} C_VEL
LIN {X 0,Y 587.424,Z 437.696,A -85,B 0,C 180,E1 -1518.649,E2 -1518.649} C_VEL
LIN {X 0,Y 587.351,Z 447.362,A -85,B 0,C 180,E1 -1519.834,E2 -1519.834} C_VEL
LIN {X 0,Y 587.266,Z 455.66,A -85,B 0,C 180,E1 -1521.05,E2 -1521.05} C_VEL
LIN {X 0,Y 587.23,Z 463.43,A -85,B 0,C 180,E1 -1522.435,E2 -1522.435} C_VEL
LIN {X 0,Y 587.18,Z 469.612,A -85,B 0,C 180,E1 -1523.816,E2 -1523.816} C_VEL
LIN {X 0,Y 587.136,Z 474.386,A -85,B 0,C 180,E1 -1525.194,E2 -1525.194} C_VEL
LIN {X 0,Y 587.18,Z 477.888,A -85,B 0,C 180,E1 -1526.569,E2 -1526.569} C_VEL
LIN {X 0,Y 587.14,Z 480.192,A -85,B 0,C 180,E1 -1527.942,E2 -1527.942} C_VEL
LIN {X 0,Y 587.135,Z 481.351,A -85,B 0,C 180,E1 -1529.314,E2 -1529.314} C_VEL
LIN {X 0,Y 587.135,Z 481.35,A -85,B 0,C 180,E1 -1530.686,E2 -1530.686} C_VEL
LIN {X 0,Y 587.14,Z 480.191,A -85,B 0,C 180,E1 -1532.058,E2 -1532.058} C_VEL
LIN {X 0,Y 587.18,Z 477.886,A -85,B 0,C 180,E1 -1533.431,E2 -1533.431} C_VEL
LIN {X 0,Y 587.136,Z 474.386,A -85,B 0,C 180,E1 -1534.806,E2 -1534.806} C_VEL
LIN {X 0,Y 587.18,Z 469.612,A -85,B 0,C 180,E1 -1536.184,E2 -1536.184} C_VEL
LIN {X 0,Y 587.23,Z 463.428,A -85,B 0,C 180,E1 -1537.565,E2 -1537.565} C_VEL
LIN {X 0,Y 587.266,Z 455.658,A -85,B 0,C 180,E1 -1538.95,E2 -1538.95} C_VEL
LIN {X 0,Y 587.351,Z 447.362,A -85,B 0,C 180,E1 -1540.166,E2 -1540.166} C_VEL
LIN {X 0,Y 587.4,Z 437.388,A -85,B 0,C 180,E1 -1541.386,E2 -1541.386} C_VEL
LIN {X 0,Y 587.521,Z 427.186,A -85,B 0,C 180,E1 -1542.434,E2 -1542.434} C_VEL
LIN {X 0,Y 587.629,Z 415.006,A -85,B 0,C 180,E1 -1543.487,E2 -1543.487} C_VEL
LIN {X 0,Y 587.753,Z 402.18,A -85,B 0,C 180,E1 -1544.408,E2 -1544.408} C_VEL
LIN {X 0,Y 587.856,Z 387.87,A -85,B 0,C 180,E1 -1545.249,E2 -1545.249} C_VEL
LIN {X 0,Y 588.028,Z 373.797,A -85,B 0,C 180,E1 -1545.911,E2 -1545.911} C_VEL
LIN {X 0,Y 588.177,Z 359.285,A -85,B 0,C 180,E1 -1546.442,E2 -1546.442} C_VEL
LIN {X 0,Y 588.256,Z 343.77,A -85,B 0,C 180,E1 -1546.857,E2 -1546.857} C_VEL
LIN {X 0,Y 588.076,Z 329.232,A -85,B 0,C 180,E1 -1547.115,E2 -1547.115} C_VEL
LIN {X 0,Y 587.259,Z 325.379,A -85,B 0,C 180,E1 -1547.204,E2 -1547.204} C_VEL
LIN {X 0,Y 587.305,Z 316.007,A -85,B 0,C 180,E1 -1549.941,E2 -1549.941} C_VEL
LIN {X 0,Y 587.342,Z 307.342,A -85,B 0,C 180,E1 -1552.514,E2 -1552.514} C_VEL
LIN {X 0,Y 587.439,Z 297.44,A -85,B 0,C 180,E1 -1555.512,E2 -1555.512} C_VEL
LIN {X 0,Y 587.502,Z 287.537,A -85,B 0,C 180,E1 -1558.588,E2 -1558.588} C_VEL
LIN {X 0,Y 587.533,Z 278.873,A -85,B 0,C 180,E1 -1561.355,E2 -1561.355} C_VEL
LIN {X 0,Y 587.651,Z 269.641,A -85,B 0,C 180,E1 -1564.391,E2 -1564.391} C_VEL
LIN {X 0,Y 587.687,Z 261.544,A -85,B 0,C 180,E1 -1567.151,E2 -1567.151} C_VEL
LIN {X 0,Y 587.764,Z 253.332,A -85,B 0,C 180,E1 -1570.07,E2 -1570.07} C_VEL
LIN {X 0,Y 587.838,Z 250.899,A -85,B 0,C 180,E1 -1571.131,E2 -1571.131} C_VEL
LIN {X 0,Y 587.693,Z 248.945,A -85,B 0,C 180,E1 -1572.146,E2 -1572.146} C_VEL
LIN {X 0,Y 587.322,Z 246.954,A -85,B 0,C 180,E1 -1573.726,E2 -1573.726} C_VEL
LIN {X 0,Y 587.306,Z 246.957,A -85,B 0,C 180,E1 -1576.883,E2 -1576.883} C_VEL
LIN {X 0,Y 587.357,Z 247.413,A -85,B 0,C 180,E1 -1577.928,E2 -1577.928} C_VEL
LIN {X 0,Y 587.327,Z 250.16,A -85,B 0,C 180,E1 -1580.639,E2 -1580.639} C_VEL
LIN {X 0,Y 587.306,Z 252.62,A -85,B 0,C 180,E1 -1583.299,E2 -1583.299} C_VEL
LIN {X 0,Y 587.22,Z 254.779,A -85,B 0,C 180,E1 -1585.771,E2 -1585.771} C_VEL
LIN {X 0,Y 587.151,Z 256.753,A -85,B 0,C 180,E1 -1588.22,E2 -1588.22} C_VEL
LIN {X 0,Y 587.159,Z 259.829,A -85,B 0,C 180,E1 -1590.901,E2 -1590.901} C_VEL
LIN {X 0,Y 587.164,Z 263.128,A -85,B 0,C 180,E1 -1593.713,E2 -1593.713} C_VEL
LIN {X 0,Y 587.128,Z 265.844,A -85,B 0,C 180,E1 -1595.985,E2 -1595.985} C_VEL
LIN {X 0,Y 587.157,Z 269.385,A -85,B 0,C 180,E1 -1598.9,E2 -1598.9} C_VEL
LIN {X 0,Y 588.277,Z 275.396,A -85,B 0,C 180,E1 -1599.029,E2 -1599.029} C_VEL
LIN {X 0,Y 588.213,Z 290.945,A -85,B 0,C 180,E1 -1599.362,E2 -1599.362} C_VEL
LIN {X 0,Y 588.142,Z 305.479,A -85,B 0,C 180,E1 -1599.816,E2 -1599.816} C_VEL
LIN {X 0,Y 587.928,Z 318.839,A -85,B 0,C 180,E1 -1600.354,E2 -1600.354} C_VEL
LIN {X 0,Y 587.845,Z 331.889,A -85,B 0,C 180,E1 -1601.018,E2 -1601.018} C_VEL
LIN {X 0,Y 587.714,Z 345.858,A -85,B 0,C 180,E1 -1601.886,E2 -1601.886} C_VEL
LIN {X 0,Y 587.621,Z 357.49,A -85,B 0,C 180,E1 -1602.762,E2 -1602.762} C_VEL
LIN {X 0,Y 587.49,Z 367.842,A -85,B 0,C 180,E1 -1603.673,E2 -1603.673} C_VEL
LIN {X 0,Y 587.398,Z 378.081,A -85,B 0,C 180,E1 -1604.739,E2 -1604.739} C_VEL
LIN {X 0,Y 587.3,Z 388.354,A -85,B 0,C 180,E1 -1606.014,E2 -1606.014} C_VEL
LIN {X 0,Y 587.272,Z 397.392,A -85,B 0,C 180,E1 -1607.385,E2 -1607.385} C_VEL
LIN {X 0,Y 587.22,Z 404.072,A -85,B 0,C 180,E1 -1608.611,E2 -1608.611} C_VEL
LIN {X 0,Y 587.185,Z 410.198,A -85,B 0,C 180,E1 -1610.006,E2 -1610.006} C_VEL
LIN {X 0,Y 587.145,Z 414.862,A -85,B 0,C 180,E1 -1611.395,E2 -1611.395} C_VEL
LIN {X 0,Y 587.151,Z 417.511,A -85,B 0,C 180,E1 -1612.434,E2 -1612.434} C_VEL
LIN {X 0,Y 587.149,Z 419.994,A -85,B 0,C 180,E1 -1613.816,E2 -1613.816} C_VEL
LIN {X 0,Y 587.125,Z 421.274,A -85,B 0,C 180,E1 -1615.194,E2 -1615.194} C_VEL
LIN {X 0,Y 587.176,Z 421.387,A -85,B 0,C 180,E1 -1616.569,E2 -1616.569} C_VEL
LIN {X 0,Y 587.139,Z 420.381,A -85,B 0,C 180,E1 -1617.942,E2 -1617.942} C_VEL
LIN {X 0,Y 587.137,Z 418.229,A -85,B 0,C 180,E1 -1619.314,E2 -1619.314} C_VEL
LIN {X 0,Y 587.141,Z 414.883,A -85,B 0,C 180,E1 -1620.686,E2 -1620.686} C_VEL
LIN {X 0,Y 587.164,Z 410.288,A -85,B 0,C 180,E1 -1622.058,E2 -1622.058} C_VEL
LIN {X 0,Y 587.199,Z 404.318,A -85,B 0,C 180,E1 -1623.431,E2 -1623.431} C_VEL
LIN {X 0,Y 587.283,Z 396.8,A -85,B 0,C 180,E1 -1624.805,E2 -1624.805} C_VEL
LIN {X 0,Y 587.316,Z 387.57,A -85,B 0,C 180,E1 -1626.183,E2 -1626.183} C_VEL
LIN {X 0,Y 587.421,Z 377.731,A -85,B 0,C 180,E1 -1627.39,E2 -1627.39} C_VEL
LIN {X 0,Y 587.523,Z 367.738,A -85,B 0,C 180,E1 -1628.426,E2 -1628.426} C_VEL
LIN {X 0,Y 587.642,Z 355.808,A -85,B 0,C 180,E1 -1629.465,E2 -1629.465} C_VEL
LIN {X 0,Y 587.763,Z 342.697,A -85,B 0,C 180,E1 -1630.42,E2 -1630.42} C_VEL
LIN {X 0,Y 587.873,Z 329.45,A -85,B 0,C 180,E1 -1631.208,E2 -1631.208} C_VEL
LIN {X 0,Y 588.008,Z 315.167,A -85,B 0,C 180,E1 -1631.899,E2 -1631.899} C_VEL
LIN {X 0,Y 588.138,Z 299.933,A -85,B 0,C 180,E1 -1632.465,E2 -1632.465} C_VEL
LIN {X 0,Y 588.235,Z 284.712,A -85,B 0,C 180,E1 -1632.879,E2 -1632.879} C_VEL
LIN {X 0,Y 588.287,Z 279.737,A -85,B 0,C 180,E1 -1632.981,E2 -1632.981} C_VEL
LIN {X 0,Y 587.899,Z 276.369,A -85,B 0,C 180,E1 -1633.12,E2 -1633.12} C_VEL
LIN {X 0,Y 586.918,Z 273.642,A -85,B 0,C 180,E1 -1633.35,E2 -1633.35} C_VEL
LIN {X 0,Y 585.601,Z 271.503,A -85,B 0,C 180,E1 -1633.642,E2 -1633.642} C_VEL
LIN {X 0,Y 583.42,Z 269.335,A -85,B 0,C 180,E1 -1634.154,E2 -1634.154} C_VEL
LIN {X 0,Y 580.824,Z 267.612,A -85,B 0,C 180,E1 -1634.943,E2 -1634.943} C_VEL
LIN {X 0,Y 580.047,Z 266.789,A -85,B 0,C 180,E1 -1635.567,E2 -1635.567} C_VEL
LIN {X 0,Y 580.037,Z 264.341,A -85,B 0,C 180,E1 -1637.633,E2 -1637.633} C_VEL
LIN {X 0,Y 580.078,Z 260.916,A -85,B 0,C 180,E1 -1640.57,E2 -1640.57} C_VEL
LIN {X 0,Y 580.093,Z 257.613,A -85,B 0,C 180,E1 -1643.566,E2 -1643.566} C_VEL
LIN {X 0,Y 580.122,Z 254.778,A -85,B 0,C 180,E1 -1646.299,E2 -1646.299} C_VEL
LIN {X 0,Y 580.095,Z 251.985,A -85,B 0,C 180,E1 -1648.987,E2 -1648.987} C_VEL
LIN {X 0,Y 580.134,Z 249.438,A -85,B 0,C 180,E1 -1651.394,E2 -1651.394} C_VEL
LIN {X 0,Y 580.172,Z 247.847,A -85,B 0,C 180,E1 -1653.033,E2 -1653.033} C_VEL
LIN {X 0,Y 580.252,Z 247.836,A -85,B 0,C 180,E1 -1655.548,E2 -1655.548} C_VEL
LIN {X 0,Y 580.286,Z 247.826,A -85,B 0,C 180,E1 -1658.147,E2 -1658.147} C_VEL
LIN {X 0,Y 580.303,Z 247.824,A -85,B 0,C 180,E1 -1660.843,E2 -1660.843} C_VEL
LIN {X 0,Y 580.242,Z 247.832,A -85,B 0,C 180,E1 -1663.662,E2 -1663.662} C_VEL
LIN {X 0,Y 580.279,Z 247.828,A -85,B 0,C 180,E1 -1666.61,E2 -1666.61} C_VEL
LIN {X 0,Y 580.297,Z 247.829,A -85,B 0,C 180,E1 -1669.156,E2 -1669.156} C_VEL
LIN {X 0,Y 580.288,Z 247.827,A -85,B 0,C 180,E1 -1671.928,E2 -1671.928} C_VEL
LIN {X 0,Y 580.256,Z 247.83,A -85,B 0,C 180,E1 -1674.453,E2 -1674.453} C_VEL
LIN {X 0,Y 580.287,Z 247.83,A -85,B 0,C 180,E1 -1676.975,E2 -1676.975} C_VEL
LIN {X 0,Y 580.298,Z 247.825,A -85,B 0,C 180,E1 -1679.425,E2 -1679.425} C_VEL
LIN {X 0,Y 580.301,Z 247.824,A -85,B 0,C 180,E1 -1682.141,E2 -1682.141} C_VEL
LIN {X 0,Y 580.275,Z 247.827,A -85,B 0,C 180,E1 -1685.281,E2 -1685.281} C_VEL
LIN {X 0,Y 580.277,Z 247.828,A -85,B 0,C 180,E1 -1687.947,E2 -1687.947} C_VEL
LIN {X 0,Y 580.285,Z 247.827,A -85,B 0,C 180,E1 -1690.913,E2 -1690.913} C_VEL
LIN {X 0,Y 580.275,Z 247.831,A -85,B 0,C 180,E1 -1693.825,E2 -1693.825} C_VEL
LIN {X 0,Y 580.328,Z 247.821,A -85,B 0,C 180,E1 -1695.983,E2 -1695.983} C_VEL
LIN {X 0,Y 580.309,Z 247.823,A -85,B 0,C 180,E1 -1698.827,E2 -1698.827} C_VEL
LIN {X 0,Y 580.331,Z 247.822,A -85,B 0,C 180,E1 -1701.644,E2 -1701.644} C_VEL
LIN {X 0,Y 580.31,Z 247.826,A -85,B 0,C 180,E1 -1704.44,E2 -1704.44} C_VEL
LIN {X 0,Y 580.347,Z 247.819,A -85,B 0,C 180,E1 -1707.918,E2 -1707.918} C_VEL
LIN {X 0,Y 580.353,Z 247.819,A -85,B 0,C 180,E1 -1710.694,E2 -1710.694} C_VEL
LIN {X 0,Y 580.28,Z 247.832,A -85,B 0,C 180,E1 -1713.472,E2 -1713.472} C_VEL
LIN {X 0,Y 580.326,Z 247.821,A -85,B 0,C 180,E1 -1715.56,E2 -1715.56} C_VEL
LIN {X 0,Y 580.307,Z 247.824,A -85,B 0,C 180,E1 -1718.356,E2 -1718.356} C_VEL
LIN {X 0,Y 580.305,Z 247.828,A -85,B 0,C 180,E1 -1721.191,E2 -1721.191} C_VEL
LIN {X 0,Y 580.317,Z 247.827,A -85,B 0,C 180,E1 -1724.017,E2 -1724.017} C_VEL
LIN {X 0,Y 580.294,Z 247.828,A -85,B 0,C 180,E1 -1726.906,E2 -1726.906} C_VEL
LIN {X 0,Y 580.289,Z 247.827,A -85,B 0,C 180,E1 -1729.823,E2 -1729.823} C_VEL
LIN {X 0,Y 580.255,Z 247.831,A -85,B 0,C 180,E1 -1732.054,E2 -1732.054} C_VEL
LIN {X 0,Y 580.309,Z 247.825,A -85,B 0,C 180,E1 -1735.08,E2 -1735.08} C_VEL
LIN {X 0,Y 580.291,Z 247.826,A -85,B 0,C 180,E1 -1738.186,E2 -1738.186} C_VEL
LIN {X 0,Y 580.275,Z 247.831,A -85,B 0,C 180,E1 -1740.692,E2 -1740.692} C_VEL
LIN {X 0,Y 580.309,Z 247.823,A -85,B 0,C 180,E1 -1743.316,E2 -1743.316} C_VEL
LIN {X 0,Y 580.232,Z 247.834,A -85,B 0,C 180,E1 -1745.754,E2 -1745.754} C_VEL
LIN {X 0,Y 580.288,Z 247.828,A -85,B 0,C 180,E1 -1748.147,E2 -1748.147} C_VEL
LIN {X 0,Y 580.301,Z 247.824,A -85,B 0,C 180,E1 -1750.844,E2 -1750.844} C_VEL
LIN {X 0,Y 580.24,Z 247.831,A -85,B 0,C 180,E1 -1753.662,E2 -1753.662} C_VEL
LIN {X 0,Y 580.282,Z 247.827,A -85,B 0,C 180,E1 -1756.609,E2 -1756.609} C_VEL
LIN {X 0,Y 580.297,Z 247.829,A -85,B 0,C 180,E1 -1759.156,E2 -1759.156} C_VEL
LIN {X 0,Y 580.291,Z 247.828,A -85,B 0,C 180,E1 -1761.928,E2 -1761.928} C_VEL
LIN {X 0,Y 580.256,Z 247.829,A -85,B 0,C 180,E1 -1764.453,E2 -1764.453} C_VEL
LIN {X 0,Y 580.287,Z 247.828,A -85,B 0,C 180,E1 -1766.975,E2 -1766.975} C_VEL
LIN {X 0,Y 580.3,Z 247.826,A -85,B 0,C 180,E1 -1769.425,E2 -1769.425} C_VEL
LIN {X 0,Y 580.295,Z 247.825,A -85,B 0,C 180,E1 -1772.143,E2 -1772.143} C_VEL
LIN {X 0,Y 580.327,Z 247.821,A -85,B 0,C 180,E1 -1775.27,E2 -1775.27} C_VEL
LIN {X 0,Y 580.275,Z 247.828,A -85,B 0,C 180,E1 -1777.947,E2 -1777.947} C_VEL
LIN {X 0,Y 580.286,Z 247.826,A -85,B 0,C 180,E1 -1780.913,E2 -1780.913} C_VEL
LIN {X 0,Y 580.275,Z 247.829,A -85,B 0,C 180,E1 -1783.825,E2 -1783.825} C_VEL
LIN {X 0,Y 580.308,Z 247.823,A -85,B 0,C 180,E1 -1785.982,E2 -1785.982} C_VEL
LIN {X 0,Y 580.312,Z 247.822,A -85,B 0,C 180,E1 -1788.827,E2 -1788.827} C_VEL
LIN {X 0,Y 580.315,Z 247.823,A -85,B 0,C 180,E1 -1791.644,E2 -1791.644} C_VEL
LIN {X 0,Y 580.306,Z 247.825,A -85,B 0,C 180,E1 -1794.44,E2 -1794.44} C_VEL
LIN {X 0,Y 580.339,Z 247.825,A -85,B 0,C 180,E1 -1797.223,E2 -1797.223} C_VEL
LIN {X 0,Y 580.357,Z 247.82,A -85,B 0,C 180,E1 -1800,E2 -1800} C_VEL
LIN {X 0,Y 580.33,Z 247.821,A -85,B 0,C 180,E1 -1802.776,E2 -1802.776} C_VEL
LIN {X 0,Y 580.32,Z 247.821,A -85,B 0,C 180,E1 -1805.56,E2 -1805.56} C_VEL
LIN {X 0,Y 580.298,Z 247.825,A -85,B 0,C 180,E1 -1808.356,E2 -1808.356} C_VEL
LIN {X 0,Y 580.306,Z 247.826,A -85,B 0,C 180,E1 -1811.191,E2 -1811.191} C_VEL
LIN {X 0,Y 580.317,Z 247.826,A -85,B 0,C 180,E1 -1814.017,E2 -1814.017} C_VEL
LIN {X 0,Y 580.318,Z 247.827,A -85,B 0,C 180,E1 -1816.913,E2 -1816.913} C_VEL
LIN {X 0,Y 580.285,Z 247.829,A -85,B 0,C 180,E1 -1819.823,E2 -1819.823} C_VEL
LIN {X 0,Y 580.254,Z 247.83,A -85,B 0,C 180,E1 -1822.053,E2 -1822.053} C_VEL
LIN {X 0,Y 580.31,Z 247.824,A -85,B 0,C 180,E1 -1825.079,E2 -1825.079} C_VEL
LIN {X 0,Y 580.25,Z 247.83,A -85,B 0,C 180,E1 -1828.188,E2 -1828.188} C_VEL
LIN {X 0,Y 580.276,Z 247.833,A -85,B 0,C 180,E1 -1830.692,E2 -1830.692} C_VEL
LIN {X 0,Y 580.305,Z 247.825,A -85,B 0,C 180,E1 -1833.316,E2 -1833.316} C_VEL
LIN {X 0,Y 580.229,Z 247.833,A -85,B 0,C 180,E1 -1835.753,E2 -1835.753} C_VEL
LIN {X 0,Y 580.292,Z 247.829,A -85,B 0,C 180,E1 -1838.146,E2 -1838.146} C_VEL
LIN {X 0,Y 580.299,Z 247.825,A -85,B 0,C 180,E1 -1840.843,E2 -1840.843} C_VEL
LIN {X 0,Y 580.247,Z 247.832,A -85,B 0,C 180,E1 -1843.661,E2 -1843.661} C_VEL
LIN {X 0,Y 580.279,Z 247.83,A -85,B 0,C 180,E1 -1846.609,E2 -1846.609} C_VEL
LIN {X 0,Y 580.306,Z 247.966,A -85,B 0,C 180,E1 -1847.237,E2 -1847.237} C_VEL
LIN {X 0,Y 580.838,Z 251.344,A -85,B 0,C 180,E1 -1848.606,E2 -1848.606} C_VEL
LIN {X 0,Y 580.783,Z 257.83,A -85,B 0,C 180,E1 -1851.005,E2 -1851.005} C_VEL
LIN {X 0,Y 580.709,Z 265.257,A -85,B 0,C 180,E1 -1853.628,E2 -1853.628} C_VEL
LIN {X 0,Y 580.643,Z 272.683,A -85,B 0,C 180,E1 -1856.167,E2 -1856.167} C_VEL
LIN {X 0,Y 580.574,Z 282.022,A -85,B 0,C 180,E1 -1859.257,E2 -1859.257} C_VEL
LIN {X 0,Y 580.483,Z 290.904,A -85,B 0,C 180,E1 -1862.107,E2 -1862.107} C_VEL
LIN {X 0,Y 580.371,Z 299.915,A -85,B 0,C 180,E1 -1864.923,E2 -1864.923} C_VEL
LIN {X 0,Y 580.303,Z 308.58,A -85,B 0,C 180,E1 -1867.574,E2 -1867.574} C_VEL
LIN {X 0,Y 580.25,Z 317.245,A -85,B 0,C 180,E1 -1870.176,E2 -1870.176} C_VEL
LIN {X 0,Y 580.228,Z 325.382,A -85,B 0,C 180,E1 -1872.582,E2 -1872.582} C_VEL
LIN {X 0,Y 581.477,Z 331.126,A -85,B 0,C 180,E1 -1872.713,E2 -1872.713} C_VEL
LIN {X 0,Y 581.414,Z 346.581,A -85,B 0,C 180,E1 -1873.008,E2 -1873.008} C_VEL
LIN {X 0,Y 581.332,Z 361.916,A -85,B 0,C 180,E1 -1873.449,E2 -1873.449} C_VEL
LIN {X 0,Y 581.119,Z 376.831,A -85,B 0,C 180,E1 -1874.03,E2 -1874.03} C_VEL
LIN {X 0,Y 580.959,Z 391.11,A -85,B 0,C 180,E1 -1874.745,E2 -1874.745} C_VEL
LIN {X 0,Y 580.8,Z 404.577,A -85,B 0,C 180,E1 -1875.58,E2 -1875.58} C_VEL
LIN {X 0,Y 580.63,Z 417.173,A -85,B 0,C 180,E1 -1876.526,E2 -1876.526} C_VEL
LIN {X 0,Y 580.515,Z 428.981,A -85,B 0,C 180,E1 -1877.591,E2 -1877.591} C_VEL
LIN {X 0,Y 580.336,Z 440.097,A -85,B 0,C 180,E1 -1878.792,E2 -1878.792} C_VEL
LIN {X 0,Y 580.27,Z 449.862,A -85,B 0,C 180,E1 -1880.061,E2 -1880.061} C_VEL
LIN {X 0,Y 580.215,Z 457.738,A -85,B 0,C 180,E1 -1881.291,E2 -1881.291} C_VEL
LIN {X 0,Y 580.13,Z 465.094,A -85,B 0,C 180,E1 -1882.692,E2 -1882.692} C_VEL
LIN {X 0,Y 580.132,Z 470.929,A -85,B 0,C 180,E1 -1884.09,E2 -1884.09} C_VEL
LIN {X 0,Y 580.041,Z 474.387,A -85,B 0,C 180,E1 -1885.135,E2 -1885.135} C_VEL
LIN {X 0,Y 580.105,Z 477.888,A -85,B 0,C 180,E1 -1886.527,E2 -1886.527} C_VEL
LIN {X 0,Y 580.039,Z 480.192,A -85,B 0,C 180,E1 -1887.917,E2 -1887.917} C_VEL
LIN {X 0,Y 580.036,Z 481.351,A -85,B 0,C 180,E1 -1889.306,E2 -1889.306} C_VEL
LIN {X 0,Y 580.036,Z 481.35,A -85,B 0,C 180,E1 -1890.694,E2 -1890.694} C_VEL
LIN {X 0,Y 580.039,Z 480.191,A -85,B 0,C 180,E1 -1892.083,E2 -1892.083} C_VEL
LIN {X 0,Y 580.105,Z 477.887,A -85,B 0,C 180,E1 -1893.473,E2 -1893.473} C_VEL
LIN {X 0,Y 580.041,Z 474.387,A -85,B 0,C 180,E1 -1894.865,E2 -1894.865} C_VEL
LIN {X 0,Y 580.093,Z 469.613,A -85,B 0,C 180,E1 -1896.26,E2 -1896.26} C_VEL
LIN {X 0,Y 580.165,Z 463.426,A -85,B 0,C 180,E1 -1897.658,E2 -1897.658} C_VEL
LIN {X 0,Y 580.207,Z 455.657,A -85,B 0,C 180,E1 -1899.06,E2 -1899.06} C_VEL
LIN {X 0,Y 580.308,Z 447.36,A -85,B 0,C 180,E1 -1900.29,E2 -1900.29} C_VEL
LIN {X 0,Y 580.383,Z 437.385,A -85,B 0,C 180,E1 -1901.525,E2 -1901.525} C_VEL
LIN {X 0,Y 580.541,Z 427.183,A -85,B 0,C 180,E1 -1902.586,E2 -1902.586} C_VEL
LIN {X 0,Y 580.678,Z 415.003,A -85,B 0,C 180,E1 -1903.651,E2 -1903.651} C_VEL
LIN {X 0,Y 580.871,Z 401.556,A -85,B 0,C 180,E1 -1904.623,E2 -1904.623} C_VEL
LIN {X 0,Y 580.997,Z 387.873,A -85,B 0,C 180,E1 -1905.434,E2 -1905.434} C_VEL
LIN {X 0,Y 581.187,Z 373.796,A -85,B 0,C 180,E1 -1906.103,E2 -1906.103} C_VEL
LIN {X 0,Y 581.352,Z 359.281,A -85,B 0,C 180,E1 -1906.64,E2 -1906.64} C_VEL
LIN {X 0,Y 581.463,Z 343.958,A -85,B 0,C 180,E1 -1907.055,E2 -1907.055} C_VEL
LIN {X 0,Y 581.374,Z 330.784,A -85,B 0,C 180,E1 -1907.296,E2 -1907.296} C_VEL
LIN {X 0,Y 580.21,Z 325.395,A -85,B 0,C 180,E1 -1907.415,E2 -1907.415} C_VEL
LIN {X 0,Y 580.243,Z 316.007,A -85,B 0,C 180,E1 -1910.194,E2 -1910.194} C_VEL
LIN {X 0,Y 580.302,Z 307.342,A -85,B 0,C 180,E1 -1912.802,E2 -1912.802} C_VEL
LIN {X 0,Y 580.403,Z 297.44,A -85,B 0,C 180,E1 -1915.844,E2 -1915.844} C_VEL
LIN {X 0,Y 580.501,Z 288.775,A -85,B 0,C 180,E1 -1918.569,E2 -1918.569} C_VEL
LIN {X 0,Y 580.552,Z 280.11,A -85,B 0,C 180,E1 -1921.369,E2 -1921.369} C_VEL
LIN {X 0,Y 580.668,Z 271.533,A -85,B 0,C 180,E1 -1924.221,E2 -1924.221} C_VEL
LIN {X 0,Y 580.741,Z 263.474,A -85,B 0,C 180,E1 -1926.992,E2 -1926.992} C_VEL
LIN {X 0,Y 580.851,Z 255.514,A -85,B 0,C 180,E1 -1929.887,E2 -1929.887} C_VEL
LIN {X 0,Y 580.863,Z 251.526,A -85,B 0,C 180,E1 -1931.718,E2 -1931.718} C_VEL
LIN {X 0,Y 580.469,Z 248.975,A -85,B 0,C 180,E1 -1933.411,E2 -1933.411} C_VEL
LIN {X 0,Y 580.267,Z 247.944,A -85,B 0,C 180,E1 -1934.626,E2 -1934.626} C_VEL
LIN {X 0,Y 580.269,Z 247.834,A -85,B 0,C 180,E1 -1936.611,E2 -1936.611} C_VEL
LIN {X 0,Y 580.342,Z 249.293,A -85,B 0,C 180,E1 -1938.662,E2 -1938.662} C_VEL
LIN {X 0,Y 580.283,Z 251.423,A -85,B 0,C 180,E1 -1940.966,E2 -1940.966} C_VEL
LIN {X 0,Y 580.233,Z 253.75,A -85,B 0,C 180,E1 -1943.594,E2 -1943.594} C_VEL
LIN {X 0,Y 580.172,Z 256.339,A -85,B 0,C 180,E1 -1946.704,E2 -1946.704} C_VEL
LIN {X 0,Y 580.078,Z 258.549,A -85,B 0,C 180,E1 -1949.413,E2 -1949.413} C_VEL
LIN {X 0,Y 580.06,Z 261.688,A -85,B 0,C 180,E1 -1952.187,E2 -1952.187} C_VEL
LIN {X 0,Y 580.071,Z 264.873,A -85,B 0,C 180,E1 -1954.909,E2 -1954.909} C_VEL
LIN {X 0,Y 580.028,Z 268.486,A -85,B 0,C 180,E1 -1957.938,E2 -1957.938} C_VEL
LIN {X 0,Y 580.054,Z 269.388,A -85,B 0,C 180,E1 -1958.686,E2 -1958.686} C_VEL
LIN {X 0,Y 581.504,Z 276.131,A -85,B 0,C 180,E1 -1958.837,E2 -1958.837} C_VEL
LIN {X 0,Y 581.398,Z 292.012,A -85,B 0,C 180,E1 -1959.191,E2 -1959.191} C_VEL
LIN {X 0,Y 581.295,Z 306.625,A -85,B 0,C 180,E1 -1959.66,E2 -1959.66} C_VEL
LIN {X 0,Y 581.077,Z 321.261,A -85,B 0,C 180,E1 -1960.28,E2 -1960.28} C_VEL
LIN {X 0,Y 580.927,Z 335.229,A -85,B 0,C 180,E1 -1961.027,E2 -1961.027} C_VEL
LIN {X 0,Y 580.77,Z 347.717,A -85,B 0,C 180,E1 -1961.844,E2 -1961.844} C_VEL
LIN {X 0,Y 580.631,Z 359.711,A -85,B 0,C 180,E1 -1962.786,E2 -1962.786} C_VEL
LIN {X 0,Y 580.463,Z 370.955,A -85,B 0,C 180,E1 -1963.831,E2 -1963.831} C_VEL
LIN {X 0,Y 580.353,Z 380.677,A -85,B 0,C 180,E1 -1964.909,E2 -1964.909} C_VEL
LIN {X 0,Y 580.261,Z 390.248,A -85,B 0,C 180,E1 -1966.16,E2 -1966.16} C_VEL
LIN {X 0,Y 580.203,Z 398.128,A -85,B 0,C 180,E1 -1967.407,E2 -1967.407} C_VEL
LIN {X 0,Y 580.12,Z 405.501,A -85,B 0,C 180,E1 -1968.823,E2 -1968.823} C_VEL
LIN {X 0,Y 580.085,Z 411.275,A -85,B 0,C 180,E1 -1970.235,E2 -1970.235} C_VEL
LIN {X 0,Y 580.084,Z 415.699,A -85,B 0,C 180,E1 -1971.641,E2 -1971.641} C_VEL
LIN {X 0,Y 580.062,Z 418.819,A -85,B 0,C 180,E1 -1973.041,E2 -1973.041} C_VEL
LIN {X 0,Y 580.089,Z 420.714,A -85,B 0,C 180,E1 -1974.438,E2 -1974.438} C_VEL
LIN {X 0,Y 580.086,Z 421.458,A -85,B 0,C 180,E1 -1975.832,E2 -1975.832} C_VEL
LIN {X 0,Y 580.035,Z 421.066,A -85,B 0,C 180,E1 -1977.222,E2 -1977.222} C_VEL
LIN {X 0,Y 580.045,Z 419.51,A -85,B 0,C 180,E1 -1978.612,E2 -1978.612} C_VEL
LIN {X 0,Y 580.041,Z 416.841,A -85,B 0,C 180,E1 -1980,E2 -1980} C_VEL
LIN {X 0,Y 580.061,Z 412.923,A -85,B 0,C 180,E1 -1981.389,E2 -1981.389} C_VEL
LIN {X 0,Y 580.071,Z 407.672,A -85,B 0,C 180,E1 -1982.778,E2 -1982.778} C_VEL
LIN {X 0,Y 580.163,Z 401.019,A -85,B 0,C 180,E1 -1984.168,E2 -1984.168} C_VEL
LIN {X 0,Y 580.239,Z 393.868,A -85,B 0,C 180,E1 -1985.386,E2 -1985.386} C_VEL
LIN {X 0,Y 580.316,Z 385.45,A -85,B 0,C 180,E1 -1986.584,E2 -1986.584} C_VEL
LIN {X 0,Y 580.425,Z 375.027,A -85,B 0,C 180,E1 -1987.829,E2 -1987.829} C_VEL
LIN {X 0,Y 580.577,Z 364.484,A -85,B 0,C 180,E1 -1988.879,E2 -1988.879} C_VEL
LIN {X 0,Y 580.728,Z 353.112,A -85,B 0,C 180,E1 -1989.843,E2 -1989.843} C_VEL
LIN {X 0,Y 580.884,Z 339.321,A -85,B 0,C 180,E1 -1990.809,E2 -1990.809} C_VEL
LIN {X 0,Y 581.015,Z 325.764,A -85,B 0,C 180,E1 -1991.588,E2 -1991.588} C_VEL
LIN {X 0,Y 581.178,Z 312.052,A -85,B 0,C 180,E1 -1992.218,E2 -1992.218} C_VEL
LIN {X 0,Y 581.39,Z 297.312,A -85,B 0,C 180,E1 -1992.745,E2 -1992.745} C_VEL
LIN {X 0,Y 581.462,Z 282.87,A -85,B 0,C 180,E1 -1993.121,E2 -1993.121} C_VEL
LIN {X 0,Y 581.338,Z 275.133,A -85,B 0,C 180,E1 -1993.274,E2 -1993.274} C_VEL
LIN {X 0,Y 580.056,Z 269.367,A -85,B 0,C 180,E1 -1993.421,E2 -1993.421} C_VEL
LIN {X 0,Y 580.047,Z 266.789,A -85,B 0,C 180,E1 -1995.567,E2 -1995.567} C_VEL
LIN {X 0,Y 579.377,Z 266.132,A -85,B 0,C 180,E1 -1996.143,E2 -1996.143} C_VEL
LIN {X 0,Y 576.51,Z 265.154,A -85,B 0,C 180,E1 -1997.078,E2 -1997.078} C_VEL
LIN {X 0,Y 574.087,Z 264.384,A -85,B 0,C 180,E1 -1997.83,E2 -1997.83} C_VEL
LIN {X 0,Y 573.044,Z 263.76,A -85,B 0,C 180,E1 -1998.411,E2 -1998.411} C_VEL
LIN {X 0,Y 572.957,Z 263.537,A -85,B 0,C 180,E1 -1998.607,E2 -1998.607} C_VEL
LIN {X 0,Y 572.986,Z 260.549,A -85,B 0,C 180,E1 -2001.221,E2 -2001.221} C_VEL
LIN {X 0,Y 573.018,Z 257.876,A -85,B 0,C 180,E1 -2003.875,E2 -2003.875} C_VEL
LIN {X 0,Y 573.051,Z 255.172,A -85,B 0,C 180,E1 -2006.454,E2 -2006.454} C_VEL
LIN {X 0,Y 573.02,Z 252.979,A -85,B 0,C 180,E1 -2008.577,E2 -2008.577} C_VEL
LIN {X 0,Y 573.054,Z 250.445,A -85,B 0,C 180,E1 -2011.004,E2 -2011.004} C_VEL
LIN {X 0,Y 573.071,Z 248.732,A -85,B 0,C 180,E1 -2012.657,E2 -2012.657} C_VEL
LIN {X 0,Y 573.203,Z 248.71,A -85,B 0,C 180,E1 -2015.188,E2 -2015.188} C_VEL
LIN {X 0,Y 573.231,Z 248.704,A -85,B 0,C 180,E1 -2017.808,E2 -2017.808} C_VEL
LIN {X 0,Y 573.249,Z 248.704,A -85,B 0,C 180,E1 -2020.525,E2 -2020.525} C_VEL
LIN {X 0,Y 573.206,Z 248.711,A -85,B 0,C 180,E1 -2023.363,E2 -2023.363} C_VEL
LIN {X 0,Y 573.244,Z 248.708,A -85,B 0,C 180,E1 -2026.332,E2 -2026.332} C_VEL
LIN {X 0,Y 573.232,Z 248.704,A -85,B 0,C 180,E1 -2028.543,E2 -2028.543} C_VEL
LIN {X 0,Y 573.237,Z 248.704,A -85,B 0,C 180,E1 -2031.298,E2 -2031.298} C_VEL
LIN {X 0,Y 573.217,Z 248.71,A -85,B 0,C 180,E1 -2034.018,E2 -2034.018} C_VEL
LIN {X 0,Y 573.234,Z 248.706,A -85,B 0,C 180,E1 -2036.515,E2 -2036.515} C_VEL
LIN {X 0,Y 573.23,Z 248.705,A -85,B 0,C 180,E1 -2039.118,E2 -2039.118} C_VEL
LIN {X 0,Y 573.242,Z 248.708,A -85,B 0,C 180,E1 -2041.436,E2 -2041.436} C_VEL
LIN {X 0,Y 573.235,Z 248.709,A -85,B 0,C 180,E1 -2044.589,E2 -2044.589} C_VEL
LIN {X 0,Y 573.24,Z 248.708,A -85,B 0,C 180,E1 -2047.662,E2 -2047.662} C_VEL
LIN {X 0,Y 573.269,Z 248.704,A -85,B 0,C 180,E1 -2050.67,E2 -2050.67} C_VEL
LIN {X 0,Y 573.248,Z 248.708,A -85,B 0,C 180,E1 -2053.622,E2 -2053.622} C_VEL
LIN {X 0,Y 573.276,Z 248.699,A -85,B 0,C 180,E1 -2055.807,E2 -2055.807} C_VEL
LIN {X 0,Y 573.267,Z 248.7,A -85,B 0,C 180,E1 -2058.745,E2 -2058.745} C_VEL
LIN {X 0,Y 573.287,Z 248.7,A -85,B 0,C 180,E1 -2061.54,E2 -2061.54} C_VEL
LIN {X 0,Y 573.279,Z 248.703,A -85,B 0,C 180,E1 -2064.372,E2 -2064.372} C_VEL
LIN {X 0,Y 573.317,Z 248.694,A -85,B 0,C 180,E1 -2067.892,E2 -2067.892} C_VEL
LIN {X 0,Y 573.325,Z 248.695,A -85,B 0,C 180,E1 -2070.702,E2 -2070.702} C_VEL
LIN {X 0,Y 573.292,Z 248.697,A -85,B 0,C 180,E1 -2072.811,E2 -2072.811} C_VEL
LIN {X 0,Y 573.293,Z 248.697,A -85,B 0,C 180,E1 -2075.628,E2 -2075.628} C_VEL
LIN {X 0,Y 573.251,Z 248.702,A -85,B 0,C 180,E1 -2078.46,E2 -2078.46} C_VEL
LIN {X 0,Y 573.277,Z 248.702,A -85,B 0,C 180,E1 -2081.312,E2 -2081.312} C_VEL
LIN {X 0,Y 573.261,Z 248.705,A -85,B 0,C 180,E1 -2084.193,E2 -2084.193} C_VEL
LIN {X 0,Y 573.254,Z 248.707,A -85,B 0,C 180,E1 -2087.112,E2 -2087.112} C_VEL
LIN {X 0,Y 573.243,Z 248.708,A -85,B 0,C 180,E1 -2090.077,E2 -2090.077} C_VEL
LIN {X 0,Y 573.223,Z 248.705,A -85,B 0,C 180,E1 -2092.339,E2 -2092.339} C_VEL
LIN {X 0,Y 573.254,Z 248.702,A -85,B 0,C 180,E1 -2095.41,E2 -2095.41} C_VEL
LIN {X 0,Y 573.229,Z 248.704,A -85,B 0,C 180,E1 -2098.565,E2 -2098.565} C_VEL
LIN {X 0,Y 573.224,Z 248.71,A -85,B 0,C 180,E1 -2100.994,E2 -2100.994} C_VEL
LIN {X 0,Y 573.267,Z 248.702,A -85,B 0,C 180,E1 -2103.524,E2 -2103.524} C_VEL
LIN {X 0,Y 573.192,Z 248.709,A -85,B 0,C 180,E1 -2106.054,E2 -2106.054} C_VEL
LIN {X 0,Y 573.243,Z 248.706,A -85,B 0,C 180,E1 -2108.702,E2 -2108.702} C_VEL
LIN {X 0,Y 573.216,Z 248.711,A -85,B 0,C 180,E1 -2111.591,E2 -2111.591} C_VEL
LIN {X 0,Y 573.217,Z 248.711,A -85,B 0,C 180,E1 -2114.674,E2 -2114.674} C_VEL
LIN {X 0,Y 573.246,Z 248.706,A -85,B 0,C 180,E1 -2117.359,E2 -2117.359} C_VEL
LIN {X 0,Y 573.235,Z 248.706,A -85,B 0,C 180,E1 -2120.392,E2 -2120.392} C_VEL
LIN {X 0,Y 573.257,Z 248.702,A -85,B 0,C 180,E1 -2123.078,E2 -2123.078} C_VEL
LIN {X 0,Y 573.257,Z 248.702,A -85,B 0,C 180,E1 -2125.67,E2 -2125.67} C_VEL
LIN {X 0,Y 573.241,Z 248.708,A -85,B 0,C 180,E1 -2128.184,E2 -2128.184} C_VEL
LIN {X 0,Y 573.269,Z 248.7,A -85,B 0,C 180,E1 -2130.634,E2 -2130.634} C_VEL
LIN {X 0,Y 573.213,Z 248.709,A -85,B 0,C 180,E1 -2133.022,E2 -2133.022} C_VEL
LIN {X 0,Y 573.28,Z 248.699,A -85,B 0,C 180,E1 -2135.366,E2 -2135.366} C_VEL
LIN {X 0,Y 573.234,Z 248.705,A -85,B 0,C 180,E1 -2138.419,E2 -2138.419} C_VEL
LIN {X 0,Y 573.275,Z 248.701,A -85,B 0,C 180,E1 -2140.731,E2 -2140.731} C_VEL
LIN {X 0,Y 573.249,Z 248.706,A -85,B 0,C 180,E1 -2143.621,E2 -2143.621} C_VEL
LIN {X 0,Y 573.254,Z 248.702,A -85,B 0,C 180,E1 -2145.806,E2 -2145.806} C_VEL
LIN {X 0,Y 573.269,Z 248.7,A -85,B 0,C 180,E1 -2148.745,E2 -2148.745} C_VEL
LIN {X 0,Y 573.259,Z 248.702,A -85,B 0,C 180,E1 -2151.54,E2 -2151.54} C_VEL
LIN {X 0,Y 573.274,Z 248.702,A -85,B 0,C 180,E1 -2154.371,E2 -2154.371} C_VEL
LIN {X 0,Y 573.317,Z 248.694,A -85,B 0,C 180,E1 -2157.892,E2 -2157.892} C_VEL
LIN {X 0,Y 573.32,Z 248.694,A -85,B 0,C 180,E1 -2160.702,E2 -2160.702} C_VEL
LIN {X 0,Y 573.299,Z 248.697,A -85,B 0,C 180,E1 -2162.81,E2 -2162.81} C_VEL
LIN {X 0,Y 573.287,Z 248.698,A -85,B 0,C 180,E1 -2165.628,E2 -2165.628} C_VEL
LIN {X 0,Y 573.243,Z 248.703,A -85,B 0,C 180,E1 -2168.46,E2 -2168.46} C_VEL
LIN {X 0,Y 573.278,Z 248.7,A -85,B 0,C 180,E1 -2171.312,E2 -2171.312} C_VEL
LIN {X 0,Y 573.272,Z 248.7,A -85,B 0,C 180,E1 -2174.418,E2 -2174.418} C_VEL
LIN {X 0,Y 573.263,Z 248.705,A -85,B 0,C 180,E1 -2177.111,E2 -2177.111} C_VEL
LIN {X 0,Y 573.24,Z 248.708,A -85,B 0,C 180,E1 -2180.077,E2 -2180.077} C_VEL
LIN {X 0,Y 573.223,Z 248.705,A -85,B 0,C 180,E1 -2182.338,E2 -2182.338} C_VEL
LIN {X 0,Y 573.248,Z 248.703,A -85,B 0,C 180,E1 -2185.41,E2 -2185.41} C_VEL
LIN {X 0,Y 573.208,Z 248.707,A -85,B 0,C 180,E1 -2188.566,E2 -2188.566} C_VEL
LIN {X 0,Y 573.223,Z 248.708,A -85,B 0,C 180,E1 -2190.993,E2 -2190.993} C_VEL
LIN {X 0,Y 573.266,Z 248.704,A -85,B 0,C 180,E1 -2193.524,E2 -2193.524} C_VEL
LIN {X 0,Y 573.254,Z 248.705,A -85,B 0,C 180,E1 -2196.922,E2 -2196.922} C_VEL
LIN {X 0,Y 573.251,Z 248.705,A -85,B 0,C 180,E1 -2199.607,E2 -2199.607} C_VEL
LIN {X 0,Y 573.221,Z 248.71,A -85,B 0,C 180,E1 -2202.639,E2 -2202.639} C_VEL
LIN {X 0,Y 573.238,Z 248.709,A -85,B 0,C 180,E1 -2205.666,E2 -2205.666} C_VEL
LIN {X 0,Y 573.265,Z 248.888,A -85,B 0,C 180,E1 -2206.916,E2 -2206.916} C_VEL
LIN {X 0,Y 573.916,Z 252.973,A -85,B 0,C 180,E1 -2208.603,E2 -2208.603} C_VEL
LIN {X 0,Y 573.821,Z 260.315,A -85,B 0,C 180,E1 -2211.344,E2 -2211.344} C_VEL
LIN {X 0,Y 573.739,Z 267.732,A -85,B 0,C 180,E1 -2213.986,E2 -2213.986} C_VEL
LIN {X 0,Y 573.643,Z 275.159,A -85,B 0,C 180,E1 -2216.542,E2 -2216.542} C_VEL
LIN {X 0,Y 573.553,Z 283.874,A -85,B 0,C 180,E1 -2219.451,E2 -2219.451} C_VEL
LIN {X 0,Y 573.445,Z 292.488,A -85,B 0,C 180,E1 -2222.243,E2 -2222.243} C_VEL
LIN {X 0,Y 573.337,Z 301.553,A -85,B 0,C 180,E1 -2225.107,E2 -2225.107} C_VEL
LIN {X 0,Y 573.263,Z 309.818,A -85,B 0,C 180,E1 -2227.663,E2 -2227.663} C_VEL
LIN {X 0,Y 573.191,Z 318.483,A -85,B 0,C 180,E1 -2230.295,E2 -2230.295} C_VEL
LIN {X 0,Y 573.163,Z 325.424,A -85,B 0,C 180,E1 -2232.373,E2 -2232.373} C_VEL
LIN {X 0,Y 574.716,Z 332.357,A -85,B 0,C 180,E1 -2232.522,E2 -2232.522} C_VEL
LIN {X 0,Y 574.635,Z 347.894,A -85,B 0,C 180,E1 -2232.834,E2 -2232.834} C_VEL
LIN {X 0,Y 574.502,Z 363.213,A -85,B 0,C 180,E1 -2233.293,E2 -2233.293} C_VEL
LIN {X 0,Y 574.287,Z 376.834,A -85,B 0,C 180,E1 -2233.835,E2 -2233.835} C_VEL
LIN {X 0,Y 574.067,Z 391.114,A -85,B 0,C 180,E1 -2234.557,E2 -2234.557} C_VEL
LIN {X 0,Y 573.888,Z 404.711,A -85,B 0,C 180,E1 -2235.411,E2 -2235.411} C_VEL
LIN {X 0,Y 573.69,Z 417.176,A -85,B 0,C 180,E1 -2236.36,E2 -2236.36} C_VEL
LIN {X 0,Y 573.528,Z 428.983,A -85,B 0,C 180,E1 -2237.437,E2 -2237.437} C_VEL
LIN {X 0,Y 573.349,Z 438.911,A -85,B 0,C 180,E1 -2238.51,E2 -2238.51} C_VEL
LIN {X 0,Y 573.273,Z 448.627,A -85,B 0,C 180,E1 -2239.76,E2 -2239.76} C_VEL
LIN {X 0,Y 573.135,Z 456.727,A -85,B 0,C 180,E1 -2241.005,E2 -2241.005} C_VEL
LIN {X 0,Y 573.093,Z 463.427,A -85,B 0,C 180,E1 -2242.247,E2 -2242.247} C_VEL
LIN {X 0,Y 573.015,Z 469.615,A -85,B 0,C 180,E1 -2243.662,E2 -2243.662} C_VEL
LIN {X 0,Y 572.951,Z 474.388,A -85,B 0,C 180,E1 -2245.074,E2 -2245.074} C_VEL
LIN {X 0,Y 573.005,Z 477.889,A -85,B 0,C 180,E1 -2246.484,E2 -2246.484} C_VEL
LIN {X 0,Y 572.938,Z 480.193,A -85,B 0,C 180,E1 -2247.891,E2 -2247.891} C_VEL
LIN {X 0,Y 572.936,Z 481.351,A -85,B 0,C 180,E1 -2249.297,E2 -2249.297} C_VEL
LIN {X 0,Y 572.936,Z 481.35,A -85,B 0,C 180,E1 -2250.703,E2 -2250.703} C_VEL
LIN {X 0,Y 572.938,Z 480.191,A -85,B 0,C 180,E1 -2252.109,E2 -2252.109} C_VEL
LIN {X 0,Y 573.005,Z 477.887,A -85,B 0,C 180,E1 -2253.516,E2 -2253.516} C_VEL
LIN {X 0,Y 572.951,Z 474.388,A -85,B 0,C 180,E1 -2254.926,E2 -2254.926} C_VEL
LIN {X 0,Y 573.014,Z 469.614,A -85,B 0,C 180,E1 -2256.338,E2 -2256.338} C_VEL
LIN {X 0,Y 573.093,Z 463.424,A -85,B 0,C 180,E1 -2257.753,E2 -2257.753} C_VEL
LIN {X 0,Y 573.135,Z 455.655,A -85,B 0,C 180,E1 -2259.173,E2 -2259.173} C_VEL
LIN {X 0,Y 573.27,Z 447.358,A -85,B 0,C 180,E1 -2260.418,E2 -2260.418} C_VEL
LIN {X 0,Y 573.358,Z 437.38,A -85,B 0,C 180,E1 -2261.669,E2 -2261.669} C_VEL
LIN {X 0,Y 573.568,Z 427.181,A -85,B 0,C 180,E1 -2262.742,E2 -2262.742} C_VEL
LIN {X 0,Y 573.728,Z 415.001,A -85,B 0,C 180,E1 -2263.82,E2 -2263.82} C_VEL
LIN {X 0,Y 573.957,Z 401.937,A -85,B 0,C 180,E1 -2264.778,E2 -2264.778} C_VEL
LIN {X 0,Y 574.123,Z 387.875,A -85,B 0,C 180,E1 -2265.623,E2 -2265.623} C_VEL
LIN {X 0,Y 574.351,Z 373.793,A -85,B 0,C 180,E1 -2266.3,E2 -2266.3} C_VEL
LIN {X 0,Y 574.529,Z 359.277,A -85,B 0,C 180,E1 -2266.844,E2 -2266.844} C_VEL
LIN {X 0,Y 574.683,Z 343.953,A -85,B 0,C 180,E1 -2267.262,E2 -2267.262} C_VEL
LIN {X 0,Y 574.603,Z 331.786,A -85,B 0,C 180,E1 -2267.491,E2 -2267.491} C_VEL
LIN {X 0,Y 573.168,Z 325.367,A -85,B 0,C 180,E1 -2267.644,E2 -2267.644} C_VEL
LIN {X 0,Y 573.245,Z 314.769,A -85,B 0,C 180,E1 -2270.827,E2 -2270.827} C_VEL
LIN {X 0,Y 573.326,Z 304.867,A -85,B 0,C 180,E1 -2273.861,E2 -2273.861} C_VEL
LIN {X 0,Y 573.416,Z 296.348,A -85,B 0,C 180,E1 -2276.528,E2 -2276.528} C_VEL
LIN {X 0,Y 573.526,Z 287.537,A -85,B 0,C 180,E1 -2279.351,E2 -2279.351} C_VEL
LIN {X 0,Y 573.625,Z 278.629,A -85,B 0,C 180,E1 -2282.287,E2 -2282.287} C_VEL
LIN {X 0,Y 573.709,Z 270.208,A -85,B 0,C 180,E1 -2285.153,E2 -2285.153} C_VEL
LIN {X 0,Y 573.833,Z 262.781,A -85,B 0,C 180,E1 -2287.762,E2 -2287.762} C_VEL
LIN {X 0,Y 573.982,Z 255.866,A -85,B 0,C 180,E1 -2290.463,E2 -2290.463} C_VEL
LIN {X 0,Y 574.007,Z 253.341,A -85,B 0,C 180,E1 -2291.68,E2 -2291.68} C_VEL
LIN {X 0,Y 573.63,Z 250.845,A -85,B 0,C 180,E1 -2293.323,E2 -2293.323} C_VEL
LIN {X 0,Y 573.378,Z 249.6,A -85,B 0,C 180,E1 -2294.691,E2 -2294.691} C_VEL
LIN {X 0,Y 573.316,Z 249.237,A -85,B 0,C 180,E1 -2296.324,E2 -2296.324} C_VEL
LIN {X 0,Y 573.361,Z 250.278,A -85,B 0,C 180,E1 -2298.393,E2 -2298.393} C_VEL
LIN {X 0,Y 573.239,Z 252.698,A -85,B 0,C 180,E1 -2301.298,E2 -2301.298} C_VEL
LIN {X 0,Y 573.179,Z 255.015,A -85,B 0,C 180,E1 -2304.024,E2 -2304.024} C_VEL
LIN {X 0,Y 573.116,Z 257.064,A -85,B 0,C 180,E1 -2306.508,E2 -2306.508} C_VEL
LIN {X 0,Y 573.043,Z 259.157,A -85,B 0,C 180,E1 -2309.15,E2 -2309.15} C_VEL
LIN {X 0,Y 572.983,Z 261.173,A -85,B 0,C 180,E1 -2311.422,E2 -2311.422} C_VEL
LIN {X 0,Y 572.989,Z 263.899,A -85,B 0,C 180,E1 -2313.797,E2 -2313.797} C_VEL
LIN {X 0,Y 572.956,Z 266.614,A -85,B 0,C 180,E1 -2316.123,E2 -2316.123} C_VEL
LIN {X 0,Y 572.961,Z 269.387,A -85,B 0,C 180,E1 -2318.464,E2 -2318.464} C_VEL
LIN {X 0,Y 574.744,Z 277.492,A -85,B 0,C 180,E1 -2318.651,E2 -2318.651} C_VEL
LIN {X 0,Y 574.575,Z 293.068,A -85,B 0,C 180,E1 -2319.016,E2 -2319.016} C_VEL
LIN {X 0,Y 574.457,Z 307.745,A -85,B 0,C 180,E1 -2319.5,E2 -2319.5} C_VEL
LIN {X 0,Y 574.194,Z 322.102,A -85,B 0,C 180,E1 -2320.128,E2 -2320.128} C_VEL
LIN {X 0,Y 574.022,Z 335.92,A -85,B 0,C 180,E1 -2320.882,E2 -2320.882} C_VEL
LIN {X 0,Y 573.815,Z 349.486,A -85,B 0,C 180,E1 -2321.801,E2 -2321.801} C_VEL
LIN {X 0,Y 573.661,Z 361.048,A -85,B 0,C 180,E1 -2322.736,E2 -2322.736} C_VEL
LIN {X 0,Y 573.46,Z 372.191,A -85,B 0,C 180,E1 -2323.811,E2 -2323.811} C_VEL
LIN {X 0,Y 573.322,Z 381.755,A -85,B 0,C 180,E1 -2324.901,E2 -2324.901} C_VEL
LIN {X 0,Y 573.214,Z 391.149,A -85,B 0,C 180,E1 -2326.168,E2 -2326.168} C_VEL
LIN {X 0,Y 573.124,Z 398.857,A -85,B 0,C 180,E1 -2327.428,E2 -2327.428} C_VEL
LIN {X 0,Y 573.048,Z 406.063,A -85,B 0,C 180,E1 -2328.856,E2 -2328.856} C_VEL
LIN {X 0,Y 573.014,Z 411.1,A -85,B 0,C 180,E1 -2330.113,E2 -2330.113} C_VEL
